# B&R Automation Studio project PLC code - cp (part 14)

#### BRSE_JSON.c
```c
/*! \file BRSE_JSON.c */
/********************************************************************
 * COPYRIGHT -- B&R
 ********************************************************************
 * Library: BRSE_JSON
 * File: BRSE_JSON.c
 * Author: Florian Damerow
 * Created: March 09, 2011
 *******************************************************************/

#include <bur/plctypes.h>
#include "BRSE_JSON.h"
#include <AsBrStr.h>
#include <string.h>
#include "BRSE_JSON_Main.h"
STRING tmpVal[80];

UDINT ValToString(UDINT pv_adresse, UINT pvType){
	switch (pvType) {
		case 1: {
				BOOL *var = (BOOL *)pv_adresse;
				brsitoa((BOOL)*var,(UDINT)&tmpVal);
				break;
				}
		case 2: {
				SINT *var = (SINT *)pv_adresse;
				brsitoa((SINT)*var,(UDINT)&tmpVal);
				break;
				}
		case 3: {
				INT *var = (INT *)pv_adresse;
				brsitoa((INT)*var,(UDINT)&tmpVal);
				break;
				}
		case 4: {
				DINT *var = (DINT *)pv_adresse;
				brsitoa((DINT)*var,(UDINT)&tmpVal);
				break;
				}
		case 5: {
				USINT *var = (USINT *)pv_adresse;
				brsitoa((USINT)*var,(UDINT)&tmpVal);
				break;
				}
		case 6: {
				UINT *var = (UINT *)pv_adresse;
				brsitoa((UINT)*var,(UDINT)&tmpVal);
				break;
				}
		case 7: {
				UDINT *var = (UDINT *)pv_adresse;
				brsitoa((UDINT)*var,(UDINT)&tmpVal);
				break;
				}
		case 8: {
				REAL *var = (REAL *)pv_adresse;
				brsftoa((REAL)*var,(UDINT)&tmpVal);
				break;
				}
		case 9: {
				STRING *var = (STRING *)pv_adresse;
				STRING *tmpBuffer = (STRING *)&tmpVal;
				strcpy(tmpVal,"\"");
				tmpBuffer++;
				strncpy(tmpBuffer,var,(sizeof(tmpVal)-3));
				strcat(tmpVal,"\"");
				break;
				}
		case 11:{
				DINT *var = (DINT *)pv_adresse;
				STRING *tmpBuffer = (STRING *)&tmpVal;
				strcpy(tmpVal,"\"");
				tmpBuffer++;
				brsitoa((DINT)*var,(UDINT)tmpBuffer);
				strcat(tmpVal,"\"");
				break;
				}
		case 12:{
				DINT *var = (DINT *)pv_adresse;
				STRING *tmpBuffer = (STRING *)&tmpVal;
				strcpy(tmpVal,"\"");
				tmpBuffer++;
				brsitoa((DINT)*var,(UDINT)tmpBuffer);
				strcat(tmpVal,"\"");
				break;
				}
		/*case 11:{
				TIME *var = pv_adresse;
				STRING *ptmpValue = &tmpValue;
				strcpy(ptmpValue,"\\/Date(");
				ptmpValue = ptmpValue + 7;
				itoa((DINT)*var,ptmpValue);
				strcat(ptmpValue,")\\/");
				break;
				}
		case 11:{
				DATE_AND_TIME *var = pv_adresse;
				BRSE_DTF_DateTimeFormat_typ format;
				UDINT error;
				error = BRSE_DTF_CreateFormat("YYYY-MM-DD-hh:mm:ss", &format);
				if(error == 0){
					BRSE_DTF_DTToString((DATE_AND_TIME)*var, &format, tmpValue);
				}
				break;
				}
		case 12:{
				TIME *var = pv_adresse;
				STRING *ptmpValue = &tmpValue;
				strcpy(ptmpValue,"\\/Time(");
				ptmpValue = ptmpValue + 7;
				itoa((DINT)*var,ptmpValue);
				strcat(ptmpValue,")\\/");
				break;
				}*/
		default: strcpy(tmpVal,"null");
				 break;
	}
	return (UDINT)tmpVal;
}

/*! \interface JSON_Parse
	\brief parses a JSON message and writes the content to the structure on the PLC

	This function block parses the JSON message and writes the content to the structure on the PLC using PV_xgetadr.\n
	The structure must exist.\n
	\n
	It is possible to parse a long JSON message in several pieces. The message can be split at every point.\n
	It is only possible to parse JSON Objects '{name:content}' \n
	arrays or non objects are NOT supported e.g. '[name:content, name2:content2]' or 'name:content' \n
	\n
	The maximal possible struture name is defined in MAX_STRUCT_NAME_LENGTH_Parse. \n
	That means the whole name e.g. 'Structure.Outer[1].Inner.Test' is limited. \n
	\n
	Entering an object will result in going up with the level by 1 \n
	Entering an array will result in going up with the level by 1 \n
	Entering an struct array will result in going up with the level by 2 \n
	\n
	If pDebug != 0 the whole message will be written there. This will be done with the state for every character.\n
	If pDebug = 0 no Debugging will be performed by the system.\n

	If pVariablesNotFound != 0 all Variables found in the Message, but could not be written on the system are listed here.
	They are represented in a JSON array e.g. '["var1","var2"]'.\n
	If pVariablesNotFound = 0 no output will performed wen variables could not be written.\n
	\n
	The funktion block will be stopped when an error accured.\n
	The function block will not be stopped when a warning accures.\n
	\par Errors:\n
	\arg 1001	invalid JSON in parsestate 0
	\arg 1002	invalid JSON in parsestate 1
	\arg 1003	invalid JSON in parsestate 3
	\arg 1004	invalid JSON in parsestate 4
	\arg 1005	invalid JSON in parsestate 6
	\arg 1006	invalid JSON in parsestate 7
	\arg 1007	Structure depth is deeper than MAX_STRUCT_DEPTH_Parse

	\par Warnings:\n
	\arg 3001	data type not supported
	\arg 3002	variable not found

	\par General: \n
	\arg 2001	parsing so far successful, but end of JSON message net reached yet
	\arg 0		successfuly finished parsing

	\param[in] pMessage Pointer to the JSON Message (String)
	\param[in] pDebug Pointer Debug Buffer (String)
	\param[in] SizeDebug size of the Debug Buffer
	\param[in] pVariablesNotFound Pointer Buffer of VariablesNotFound (String)
	\param[in] SizeVariablesNotFound size of the VariablesNotFound Buffer
	\param[in] MaxLoopIdx used to control cpu load. Allows multiple entries to be parsed each scan.

	\param[out] ErrorInfo contains the Error/Warning/General Codes.
	\param[out] Status signals when block is done=1 or error=2.

*/

void JSON_Parse(struct JSON_Parse* inst)
{
	STRING *pBuff = (STRING *)inst->pMessage;

	UDINT pBuffOld = 0;
	inst->ErrorInfo = 0;

	/* gets the length of the message, only 1 time */
	if(inst->messageLength == 0) {
		inst->messageLength = brsstrlen((UDINT)inst->pMessage);
	}

	if(inst->MaxLoopIdx == 0) {
		inst->MaxLoopIdx = 1000;					// try to set a default value
	}

	/* 	loop index makes it possible to process larger strings, since we don't have to process the whole string in 1 cycle.
			We try to process mutiple variables in 1 cycle.
			If max. loop index is too high we get a cycle time violation.
	*/
	while(inst->buffIdx < inst->messageLength && inst->loopIdx < inst->MaxLoopIdx){			/* while buffer indeex is smaller than length and loop index smaller then max loop index */
		switch(inst->parsestate){
			case 0:
				if(pBuff[inst->buffIdx] == '{'){
					inst->parsestate = 1;
					inst->parselevel++;
					inst->buffIdx++;
					if(inst->pVariablesNotFound != 0 && inst->SizeVariablesNotFound > 2){
						strcpy((STRING *)inst->pVariablesNotFound,"[");
					}
				}
				else if(pBuff[inst->buffIdx] == ' '){
					inst->buffIdx++;
				}
				else{
					inst->ErrorInfo = 1001; /*invalid JSON*/
					inst->Status 	= 2;
					return;
				}
				break;

			case 1:
				if(pBuff[inst->buffIdx] == '"'){
					inst->parsestate = 2;
					inst->buffIdx++;
				}
				else if(pBuff[inst->buffIdx] == ' ' || pBuff[inst->buffIdx] == 9 || pBuff[inst->buffIdx] == 10 || pBuff[inst->buffIdx] == 11 || pBuff[inst->buffIdx] == 12){
					inst->buffIdx++;
				}
				else{
					inst->ErrorInfo = 1002; /*invalid JSON*/
					inst->Status 	= 2;
					return;
				}
				break;

			case 2:
				if(pBuff[inst->buffIdx] != '"'){
					inst->pvName[inst->parselevel][inst->j] = pBuff[inst->buffIdx];
					inst->j++;
					inst->buffIdx++;
				}
				else {
					inst->pvName[inst->parselevel][inst->j] = '\0';
					inst->j = 0;
					inst->parsestate = 3;
					inst->buffIdx++;
				}
				break;

			case 3:
				if(pBuff[inst->buffIdx] == ':'){
					inst->parsestate = 4;
					inst->buffIdx++;
				}
				else if(pBuff[inst->buffIdx] == ' ' || pBuff[inst->buffIdx] == 9 || pBuff[inst->buffIdx] == 10 || pBuff[inst->buffIdx] == 11 || pBuff[inst->buffIdx] == 12){
					inst->buffIdx++;
				}
				else{
					inst->ErrorInfo = 1003; /*invalid JSON*/
					inst->Status 	= 2;
					return;
				}
				break;

			case 4:
				if(pBuff[inst->buffIdx] == '{'){
					inst->parsestate = 1;
					inst->parselevel++;
					inst->buffIdx++;
				}
				else if(pBuff[inst->buffIdx] == '['){
					/*strcat(inst->pvName[inst->parselevel],"[");
					strcat(inst->pvName[inst->parselevel],"0");
					strcat(inst->pvName[inst->parselevel],"]");*/
					inst->isArray[inst->parselevel] = 1;
					inst->parselevel++;
					inst->buffIdx++;
				}
				else if(pBuff[inst->buffIdx] == '\"'){
					inst->Buffer[inst->j] = pBuff[inst->buffIdx];
					inst->buffIdx++;
					inst->j++;
					inst->parsestate = 41;
				}
				else if(pBuff[inst->buffIdx] != '{' && pBuff[inst->buffIdx] != ' ' && pBuff[inst->buffIdx] != '['){ /*maybe better to check for " or - or number*/
					inst->parsestate = 5;
				}
				else if(pBuff[inst->buffIdx] == ' ' || pBuff[inst->buffIdx] == 9 || pBuff[inst->buffIdx] == 10 || pBuff[inst->buffIdx] == 11 || pBuff[inst->buffIdx] == 12){
					inst->buffIdx++;
				}
				else{
					inst->ErrorInfo = 1004; /*invalid JSON*/
					inst->Status 	= 2;
					return;
				}
				break;

			case 41: /* is in String */
				if(pBuff[inst->buffIdx] == '\"'){
					inst->Buffer[inst->j] = pBuff[inst->buffIdx];
					inst->j++;
					inst->Buffer[inst->j] = '\0';
					inst->j=0;
					inst->buffIdx++;
					inst->parsestate = 51;
				}
				else if(pBuff[inst->buffIdx] == '\\'){
					inst->Buffer[inst->j] = pBuff[inst->buffIdx];
					inst->j++;
					inst->buffIdx++;
					inst->Buffer[inst->j] = pBuff[inst->buffIdx];
					inst->j++;
					inst->buffIdx++;
				}
				else{
					inst->Buffer[inst->j] = pBuff[inst->buffIdx];
					inst->j++;
					inst->buffIdx++;
				}
				break;

			case 5:
				if(pBuff[inst->buffIdx] != '}' && pBuff[inst->buffIdx] != ' ' && pBuff[inst->buffIdx] != ',' && pBuff[inst->buffIdx] != ']'){
					inst->Buffer[inst->j] = pBuff[inst->buffIdx];
					inst->j++;
					inst->buffIdx++;
				}
				else{
					STRING mystring[5] = "256";

					UINT myint = strcmp(mystring, inst->Buffer);
					if(myint == 0)
					{
						inst->j = inst->j;
					}
					inst->Buffer[inst->j] = '\0';
					inst->j=0;
					inst->parsestate = 51;
				}
				break;

			case 51: /*write variable*/
				memset((UDINT *)(inst->fullName),0,sizeof(inst->fullName));
				{
					UINT i = 1;
					UDINT adresse;
					UDINT datalen;
					UDINT pvType;
					UDINT pvLength;
					UINT pvStructMembers;
					STRING tmpStr[5];
					while(i <= inst->parselevel && (sizeof(inst->fullName)-strlen(inst->fullName)-7) > strlen(inst->pvName[i])){
						strcat(inst->fullName,inst->pvName[i]);
						if(inst->isArray[i] == 1){
							strcat(inst->fullName,"[");
							brsitoa(inst->pvIndex[i],(UDINT)&tmpStr);
							strcat(inst->fullName,tmpStr);
							strcat(inst->fullName,"]");
						}
						if(i < inst->parselevel && inst->isArray[i] == 0){
							strcat(inst->fullName,".");
						}
						i++;
					}
					inst->ErrorInfo = PV_ninfo((STRING *)&inst->fullName, &pvType, &pvLength, &pvStructMembers);
					if(inst->ErrorInfo == 0){
						inst->ErrorInfo = PV_xgetadr((STRING *)&inst->fullName, &adresse, &datalen);
					}
					else{
						inst->ErrorInfo = 3002; /* variable not found */
					}
					if(inst->ErrorInfo == 0){
						STRING *Buffer = (STRING *)&inst->Buffer;
						if(*Buffer == '\"'){
							Buffer++;
							if(inst->Buffer[strlen(Buffer)] == '\"'){
								inst->Buffer[strlen(Buffer)] = '\0';
							}
						}
						if(strstr(inst->Buffer,"null") == 0){
							switch(pvType){
								case 0:{
									DINT *adr = (DINT *)adresse;
									*adr = (DINT)brsatoi((UDINT)Buffer);
									break;
									}
								case 1:{
										BOOL *adr = (BOOL *)adresse;

										if(strstr(Buffer, "true")){
											*adr = 1;
										}
										else if(strstr(Buffer, "false")){
											*adr = 0;
										}
										else if(brsatoi((UDINT)Buffer) != 0){
											*adr = 1;
										}
										else{
											*adr = 0;
										}
										break;
									}
								case 2:{
									SINT *adr = (SINT *)adresse;
									*adr = (SINT)brsatoi((UDINT)Buffer);
									break;
									}
								case 3:{
									INT *adr = (INT *)adresse;
									*adr = (INT)brsatoi((UDINT)Buffer);
									break;
									}
								case 4:{
									DINT *adr = (DINT *)adresse;
									*adr = (DINT)brsatoi((UDINT)Buffer);
									break;
									}
								case 5:{
									USINT *adr = (USINT *)adresse;
									*adr = (USINT)brsatoi((UDINT)Buffer);
									break;
									}
								case 6:{
									UINT *adr = (UINT *)adresse;
									*adr = (UINT)brsatoi((UDINT)Buffer);
									break;
									}
								case 7:{
									UDINT *adr = (UDINT *)adresse;
									*adr = (UDINT)brsatoi((UDINT)Buffer);
									break;
									}
								case 8:{
									REAL *adr = (REAL *)adresse;
									*adr = (REAL)brsatof((UDINT)Buffer);
									break;
									}
								case 9:{
									STRING *adr = (STRING *)adresse;
									strncpy(adr, Buffer, pvLength-1);
									break;
									}
								case 11:{
									DINT *adr = (DINT *)adresse;
									*adr = (DINT)brsatoi((UDINT)Buffer);
									break;
									}
								case 12:{
									DINT *adr = (DINT *)adresse;
									*adr = (DINT)brsatoi((UDINT)Buffer);
									break;
									}
								case 14:{
										LREAL *adr = (LREAL *)adresse;
										*adr = (LREAL)brsatof((UDINT)Buffer);
										break;
									}
								/*case 11:{
									DINT *adr = adresse;
									STRING *Buffer = &inst->Buffer;
									Buffer = strstr(inst->Buffer,")\\/");
									if(Buffer != 0){
										*Buffer = '\0';
										Buffer = strstr(inst->Buffer,"\\/Date(");
										if(Buffer != 0){
											Buffer = Buffer + 7;
										}
									}
									*adr = (DINT)atoi(Buffer);
									break;
									}
								case 12:{
									DINT *adr = adresse;
									STRING *Buffer = &inst->Buffer;
									Buffer = strstr(inst->Buffer,")\\/");
									if(Buffer != 0){
										*Buffer = '\0';
										Buffer = strstr(inst->Buffer,"\\/Time(");
										if(Buffer != 0){
											Buffer = Buffer + 7;
										}
									}
									*adr = (DINT)atoi(Buffer);
									break;
									}*/

								default:{
									inst->ErrorInfo = 3001;
									break;
									}
							}
						}
					}
					else{
						inst->ErrorInfo = 3002; /* variable not found */
						if(inst->pVariablesNotFound != 0 && inst->SizeVariablesNotFound != 0){
							if((inst->SizeVariablesNotFound - strlen((STRING *)inst->pVariablesNotFound)-2) > strlen(inst->fullName)+3){
								if(strlen((STRING *)inst->pVariablesNotFound) > 2){
									strcat((STRING *)inst->pVariablesNotFound,",");
								}
								strcat((STRING *)inst->pVariablesNotFound,"\"");
								strcat((STRING *)inst->pVariablesNotFound,inst->fullName);
								strcat((STRING *)inst->pVariablesNotFound,"\"");
							}
						}
					}
					if(pBuff[inst->buffIdx] == ',' && inst->isArray[inst->parselevel-1] == 1){
						inst->buffIdx++;
						inst->pvIndex[inst->parselevel-1]++;
						inst->parsestate = 4;
					}
					else{
						inst->parsestate = 6;
					}
				}
				break;

			case 6:
				if(pBuff[inst->buffIdx] == '}'){
					inst->parsestate = 6;
					inst->pvIndex[inst->parselevel-1] = 0;
					strcpy(inst->pvName[inst->parselevel],"");	// if the string is not cleared, the parseing is not working right - olsenm
					inst->parselevel--;
					inst->buffIdx++;
				}
				else if(pBuff[inst->buffIdx] == ']'){
					inst->parsestate = 6;
					inst->pvIndex[inst->parselevel-1] = 0;
					strcpy(inst->pvName[inst->parselevel],"");	// if the string is not cleared, the parseing is not working right - olsenm
					inst->parselevel--;
					inst->isArray[inst->parselevel] = 0;
					inst->buffIdx++;
				}
				else if(pBuff[inst->buffIdx] == ','){
					inst->parsestate = 7;
					inst->pvIndex[inst->parselevel-1]++;
					inst->buffIdx++;
				}
				else if(pBuff[inst->buffIdx] == ' ' || pBuff[inst->buffIdx] == 9 || pBuff[inst->buffIdx] == 10 || pBuff[inst->buffIdx] == 11 || pBuff[inst->buffIdx] == 12){
					inst->buffIdx++;
				}
				else{
					inst->ErrorInfo = 1005; /*invalid JSON*/
					inst->Status 	= 2;
					return;
				}
				break;

			case 7:
				if(pBuff[inst->buffIdx] == '{'){
					inst->parselevel++;
					inst->parsestate = 1;
					inst->buffIdx++;
				}
				else if(pBuff[inst->buffIdx] == '\"'){
					inst->parsestate = 1;
				}
				else if(pBuff[inst->buffIdx] == ' ' || pBuff[inst->buffIdx] == 9 || pBuff[inst->buffIdx] == 10 || pBuff[inst->buffIdx] == 11 || pBuff[inst->buffIdx] == 12){
					inst->buffIdx++;
				}
				else{
					inst->ErrorInfo = 1006; /*invalid JSON*/
					inst->Status 	= 2;
					return;
				}
		}

		/* DEBUGGING */
		if(inst->pDebug != 0){
			if(pBuffOld != pBuff[inst->buffIdx]){
				STRING BUFFER2[4];
				STRING BUFFER3[2];
				if((inst->SizeDebug - strlen((STRING *)inst->pDebug) - 1) > 7){
					if(inst->parsestateold != inst->parsestate){
						inst->parsestateold = inst->parsestate;
						brsitoa((DINT)inst->parsestate,(UDINT)&BUFFER2);
						strcat((STRING *)inst->pDebug,"(");
						strcat((STRING *)inst->pDebug,BUFFER2);
						strcat((STRING *)inst->pDebug,")");
					}
					BUFFER3[0] = pBuff[inst->buffIdx];
					BUFFER3[1] = 0;
					strcat((STRING *)inst->pDebug,BUFFER3);
				}
			}
			pBuffOld = pBuff[inst->buffIdx];
		}
		inst->loopIdx++;			// loop index counter
	}
	inst->loopIdx = 0;		// reset loop index

	/* Error Handling */
	if(inst->parselevel > MAX_STRUCT_DEPTH_Parse){
		inst->ErrorInfo = 1007;
	}
	if(inst->ErrorInfo >= 1000 && inst->ErrorInfo  < 2000){
		inst->parselevel = 0;
		inst->parsestate = 0;
		memset(inst->pvIndex,0,sizeof(inst->pvIndex));
		memset(inst->pvName,0,sizeof(inst->pvName));
	}
	else if(inst->parselevel != 0){
		inst->ErrorInfo = 2001; /*not done*/
	}
	else{
		if(inst->pVariablesNotFound != 0){
			strcat((STRING *)inst->pVariablesNotFound,"]");
		}
		inst->parsestate = 0;
	}

	/*Status output*/
	if(inst->buffIdx >= inst->messageLength)
	{
		if(inst->ErrorInfo > 0)
		{
			//Done, Error present.
			inst->Status = 2;
		}
		else
		{
			//Done, no errors present.
			inst->Status = 1;
		}

	}
}

/*! \interface JSON_Stringify
	\brief converts a PV variable and the whole structure into a JSON Object using PV_ninfo.

	This function block converts the whole structure of a PV variable into a JSON Object using PV_ninfo. \n
	The variable name should be the same as using the PV_ninfo function. By that it is possible to access any kind of PV variables.\n
	The output is always a JSON object. e.g. '{"varname": ... }' \n
	\n
	The function block has to be run several times until the Status = 1. \n
	Every time the function block is called it creates the JSON output for one new variable inside the Structure. \n
	If the variable in the structure is an array of a non object type the whole array will be created in Output.\n
	\n
	The maximum Output length is defined by MAX_OUTPUT_LENGTH_Stringify.\n
	The maximum Value of a nun array, non structure variable is 80. So Strings are only supported up the 80 characters.\n
	\n
	By using pMessage and MaxLoopIndex multiple entries can be stringified in one scan.\n
	The complete json string is written directly to the buffer pMessage is pointing to.\n

	\par Status Codes:\n
	\arg 1001 Variable not found
	\arg 1002 Variable value too long
	\arg 1003 pStName = 0, zero pointer
	\arg 1 stringify process completed
	\arg 0 stringify process not completet yet - run again

	\param[in] pStName Pointer to the requested variable name
	\param[in] pMessage pointer to output buffer where the entire JSON_String is written.
	\param[in] MaxLoopIndex used to control cpu load. Allows multiple entries to be stringified each scan.

	\param[out] Status returns the Status codes
	\param[out] Output contains the content of one step

*/
void JSON_Stringify(struct JSON_Stringify* inst)
{
	/*
			the loop index makes it possible to process mutiple variables in one cycle
			if the maxloopisx is too high we get a cycle time violation
	*/

	if(inst->MaxLoopIdx == 0) {
		inst->MaxLoopIdx = 100;			// default value
	}

	memset(inst->Output,0,sizeof(inst->Output));

	for(inst->loopIdx = 0; inst->loopIdx < inst->MaxLoopIdx; inst->loopIdx++) {
		STRING *pBuff = 0;
		STRING strBuff[20];
		inst->TaskDoc.Input.StructDepth = MAX_STRUCT_DEPTH_Stringify;

		/*gather information of the structure item*/
		memset(inst->tmpStruct,0,sizeof(inst->tmpStruct));

		if(inst->pStName != 0 )
		{
			strcpy(inst->tmpStruct,(STRING *)inst->pStName);
		}
		else
		{
			inst->Status = 1003;
			return;
		}

		strcat(inst->tmpStruct, inst->pvName[0]);
		for( inst->i = 1; inst->i <= inst->pvLevel; inst->i++ ){
			if(inst->isArray[inst->i-1] == 0){
				strcat(inst->tmpStruct, ".");
				strcat(inst->tmpStruct, inst->pvName[inst->i]);
			}
			else{
				inst->isArray[inst->pvLevel] = 1;
				strcat(inst->tmpStruct,"[");
				brsitoa(inst->pvIndex[inst->i-1],(UDINT)&strBuff);
				strcat(inst->tmpStruct,strBuff);
				strcat(inst->tmpStruct,"]");
			}
		}
		/*Search in PV-list*/
		inst->TaskDoc.Output.StatusInfo = PV_ninfo((STRING *)&inst->tmpStruct, &inst->pvType, &inst->pvLength, &inst->pvStructMembers[inst->pvLevel]);
		if(inst->pvType == 0){
			STRING name[80];
			inst->TaskDoc.Output.StatusSearch = PV_item((STRING *)&inst->tmpStruct, 0, (STRING *)&name);
			if(inst->TaskDoc.Output.StatusSearch != 0){
				inst->pvType = 4;
				inst->pvStructMembers[inst->pvLevel] = 1;
				inst->TaskDoc.Output.StatusSearch = 0;
			}
		}
		if(inst->pvType == 15){
			inst->isArray[inst->pvLevel] = 1;
			strcat(inst->tmpStruct,"[");
			brsitoa(inst->pvIndex[inst->pvLevel],(UDINT)&strBuff);
			strcat(inst->tmpStruct,strBuff);
			strcat(inst->tmpStruct,"]");
			inst->pvLevel = inst->pvLevel + 1;
			inst->TaskDoc.Output.StatusInfo = PV_ninfo((STRING *)&inst->tmpStruct, &inst->pvType, &inst->pvLength, &inst->pvStructMembers[inst->pvLevel]);
		}
		else{
			inst->isArray[inst->pvLevel] = 0;
		}
		if( inst->TaskDoc.Output.StatusInfo == 0 ){
			inst->TaskDoc.Output.StatusInfo = PV_xgetadr((STRING *)&inst->tmpStruct,&inst->pv_adresse,&inst->data_len);
		}
		if( inst->TaskDoc.Output.StatusInfo == 0 ){
		/*variable was found*/
			STRING *ValToStr;
			UDINT Size=0;
			memset(inst->tmpValue,0,sizeof(inst->tmpValue));
			if(inst->pvStructMembers[inst->pvLevel]>1){
				strcat(inst->tmpValue,"[");
			}
			ValToStr = (STRING *)ValToString(inst->pv_adresse, inst->pvType);
			if((sizeof(inst->tmpValue)-strlen(inst->tmpValue)-2) > strlen(ValToStr)){
				strcat(inst->tmpValue, ValToStr);
			}
			inst->arrIndex = 1;
			Size = (UDINT)(inst->data_len/inst->pvStructMembers[inst->pvLevel]);
			pBuff = (STRING *)((UDINT)inst->pv_adresse+Size);
			/*build array output */
			while(inst->arrIndex < inst->pvStructMembers[inst->pvLevel]){
				ValToStr = (STRING *)ValToString((UDINT)pBuff, inst->pvType);
				if((sizeof(inst->tmpValue)-strlen(inst->tmpValue)-2) <= strlen(ValToStr)){
					inst->Status = 1002; /*Variable Value too long*/
					return;
				}
				strcat(inst->tmpValue, ",");
				strcat(inst->tmpValue, ValToStr);
				pBuff = pBuff+Size;
				inst->arrIndex++;
			}
			if(inst->pvStructMembers[inst->pvLevel]>1){
				strcat(inst->tmpValue,"]");
			}

			/*get inner variable name*/
			pBuff = (inst->tmpStruct)+strlen(inst->tmpStruct);
			while((UDINT)pBuff >= (UDINT)&(inst->tmpStruct) && *pBuff != '.'){
				pBuff--;
			}
			pBuff++;
			/*create JSON output*/
			//memset(inst->Output,0,sizeof(inst->Output)); Memset should be done outside for loop. Or output will just contain the latest iteration output. Valdtp V1.11.0
			if((43+strlen(inst->tmpValue)) > sizeof(inst->Output)){
				inst->Status = 1002; /*Variable Value too long*/
				return;
			}
			if(!(inst->isArray[inst->pvLevel-1] == 1 && inst->pvIndex[inst->pvLevel-1] > 0)){
				if((inst->pvLevel == 0 && inst->pvIndex[0] == 0) || (inst->isArray[inst->pvLevel-1] == 1 && (inst->pvLevel-1) == 0) ){
					strcat(inst->Output, "{");

				}
				strcat(inst->Output, "\"");
				if( inst->pvLevel == 0){
					strcat(inst->Output, (STRING *)inst->pStName);
				}
				else if(inst->isArray[inst->pvLevel-1] == 1){
					if((inst->pvLevel-1) > 0){
						strcat(inst->Output, inst->pvName[inst->pvLevel-1]);
					}
					else{
						strcat(inst->Output, (STRING *)inst->pStName);
					}
				}else{
					strcat(inst->Output, inst->pvName[inst->pvLevel]);
				}
				strcat(inst->Output, "\":");
				if(inst->isArray[inst->pvLevel-1]){
					strcat(inst->Output, "[");
				}
			}
			if( inst->pvType == 0 ){
				strcat(inst->Output, "{");
			}
			if( inst->pvType != 0 && inst->pvType != 15 ){
				strcat(inst->Output, inst->tmpValue);
			}

			inst->pvSearchComplete = 0;

			if( (inst->pvType == 0) && (inst->pvLevel < (inst->TaskDoc.Input.StructDepth-1)) ){
				/*variable is a structure and its ok to go look inside it*/
				/*ok. proceed to next level.*/
				inst->TaskDoc.Output.StatusSearch = PV_item((STRING *)&inst->tmpStruct, inst->pvIndex[inst->pvLevel], (STRING *)&inst->pvName[inst->pvLevel+1]);
				inst->pvLevel = inst->pvLevel + 1;
			}
			else if( (inst->pvLevel > 0) || (inst->pvLevel==0 && inst->pvIndex[inst->pvLevel] < (inst->pvStructMembers[inst->pvLevel]))){ /*..in case its 0 we have a problem*/
			/*variable is a basic datatype*/
				do{
					inst->pvContinue = 0;
					if( inst->isArray[inst->pvLevel-1] == 1){
						if( inst->pvIndex[inst->pvLevel-1] < (inst->pvStructMembers[inst->pvLevel-1]-1)){
							/*ok. take the next item in prior structure*/
							inst->pvIndex[inst->pvLevel-1] = inst->pvIndex[inst->pvLevel-1] + 1;
							strcpy(inst->pvName[inst->pvLevel],"");		// if the string is not cleared, the stringify is not working right - olsenm
							inst->pvLevel = inst->pvLevel - 1;

							strcat(inst->Output, ",");
							break; /*..from loop*/
						}
						else{
							strcat(inst->Output, "]");
							strcpy(inst->pvName[inst->pvLevel],"");		// if the string is not cleared, the stringify is not working right - olsenm
							inst->pvLevel = inst->pvLevel - 1;
							inst->pvIndex[inst->pvLevel] = 0;
							if( inst->pvLevel > 0 ){
								inst->pvContinue = 1;
							}else{
								inst->pvSearchComplete = 1;
								strcat(inst->Output, "}");
								break;
							}
						}
					}
					else{
						if( inst->pvIndex[inst->pvLevel-1] < (inst->pvStructMembers[inst->pvLevel-1]-1)){
							/*ok. take the next item in prior structure*/
							inst->pvIndex[inst->pvLevel-1] = inst->pvIndex[inst->pvLevel-1] + 1;
							strcat(inst->Output, ",");
							break; /*..from loop*/
						}else{
							/*continue looking in the prior structure if the index is smaller members*/
							strcpy(inst->pvName[inst->pvLevel],"");																		// if the string is not cleared, the stringify is not working right - olsenm
							inst->pvLevel = inst->pvLevel - 1;
							if(inst->pvLevel>=0){
								strcat(inst->Output, "}");
							}
							inst->pvIndex[inst->pvLevel] = 0; /*this one is used the nest time a structure is found on this level*/
							if( inst->pvLevel > 0 ){
								inst->pvContinue = 1;
							}else{
								inst->pvSearchComplete = 1;
								strcat(inst->Output, "}");
								break;
							}
						}
					}
				}
				while(inst->pvContinue != 0);

				/*look after following member in prior structure*/
				if( inst->pvLevel > 0 ){
					strcpy(inst->tmpStruct,(STRING *)inst->pStName);

					strcat(inst->tmpStruct, inst->pvName[0]);
					for( inst->i = 1; inst->i <= (inst->pvLevel-1); inst->i++ ){
						if(strlen(inst->pvName[inst->i]) != 0){
							strcat(inst->tmpStruct, ".");
							strcat(inst->tmpStruct, inst->pvName[inst->i]);
						}
					}
					/*ok. get the next variable*/
					inst->TaskDoc.Output.StatusSearch = PV_item((STRING *)&inst->tmpStruct, inst->pvIndex[inst->pvLevel-1], (STRING *)&inst->pvName[inst->pvLevel]);
				}else if((inst->pvLevel==0 && inst->pvIndex[inst->pvLevel] == (inst->pvStructMembers[inst->pvLevel]))){
					/*no more items in top structure*/
					inst->pvSearchComplete = 1;
				}
			}else{
				inst->pvSearchComplete = 1;
			}
			if(inst->pvSearchComplete == 1){
				inst->Status = 1;
			}else{
				inst->Status = 0;
			}
		}else{
			 inst->Status = 1001; /*variable not found*/
		}

		if(inst->Status == 1) {
			break; 									// break out of for loop because the function block is done processing the variables
		}

	}//END FOR

	/*Must always check that pointers are != 0 or it will krasch PLC. Valdtp V1.11.0*/
	if(inst->pMessage != 0)
	{
		/*
			instead of copying the output outside the fb we do in inside, so we can process mutiple variables in 1 cycle  -olsenm
		*/
		UDINT outLen = brsstrlen((UDINT)inst->Output);// length of the generated output string
		UDINT tmpMsgPtr = (UDINT)&((char*)inst->pMessage)[inst->messageIdx];	// pointer to where the output can be copied to
		strcpy((char*)tmpMsgPtr,inst->Output);									// copy the string
		inst->messageIdx += outLen;		// messageidx keeps track of where in the message string we can copy the output string

	}

}
```

#### version_history.c
```c
/*!\file version_history.c */

/*!
	\page History
	\section History

	\par V1.00.0
		\arg First version created

	\par V1.00.1
		\arg Helpfile and example added.

	\par V1.01.0
		\arg Helpfile updated
		\arg First release version.

	\par V1.02.0
		\arg Helpfile updated

	\par V1.10.0
		\arg Library dependency changed from AsString to AsBrStr.
             Add #include <AsBrStr.h>
        \arg Functions atof, ftoa, atoi and itoa are changed to brsatof, brsftoa, brsatoi, and brsitoa
             to avoid name conflict.
        \arg Functions strcat and strcpy can continue to be used from string.h
	\par V1.11.0
		\arg Library updated, changed command structure for functions. Improving usage with large data amounts.
			 Possible to set number of iterations run per scan.
			 Output directly into an output buffer has beeen added making it possible to stringify several entries in one scan.

		\arg Examples replaced and simplified. Package that is imported instead of an entire project.
			 The simplification should make the javascript code and example tasks easier to understand.
			 TestProgram task added.
	\par V1.12.0
		\arg Added support for ASCII charaters 9 -> 12. TAB, New Line, Vertical Tab and New page.
			 Have the same effect has an blank space ' '.
			 This to ease the usage of third party software like Notepad++ for editing of the JSON string.
*/
```

### MTFilter.var
```iecst
(*Error*)
VAR CONSTANT
	mtBCD_ERR_FILTER_TYPE_INVALID : DINT := -1058012158; (*Filter type is invalid.*)
	mtBCD_ERR_FILTER_ORDER_INVALID : DINT := -1058012157; (*Filter order is invalid.*)
	mtBCD_ERR_CUTOFF_FREQ_INVALID : DINT := -1058012156; (*Cutoff frequency of the filter is invalid.*)
	mtBCD_ERR_CENTER_FREQ_INVALID : DINT := -1058012155; (*Center frequency of the filter is invalid.*)
	mtBCD_ERR_FILTER_BANDWIDTH : DINT := -1058012154; (*Bandwidth of the filter is invalid.*)
	mtBCD_ERR_FREQ_NUM_INVALID : DINT := -1058012153; (*Filter frequency of the numerator is invalid.*)
	mtBCD_ERR_DAMPING_NUM_INVALID : DINT := -1058012152; (*Damping of the numerator is invalid.*)
	mtBCD_ERR_FREQ_DEN_INVALID : DINT := -1058012151; (*Filter frequency of the denominator is invalid.*)
	mtBCD_ERR_DAMPING_DEN_INVALID : DINT := -1058012150; (*Damping of the denominator is invalid.*)
	mtBCD_ERR_FILTER_WINDOW_INVALID : DINT := -1058012149; (*Window length of the filter is invalid.*)
	mtBCD_ERR_TRANSFER_FCN_INVALID : DINT := -1058012148; (*Transfer function (Numerator or Denominator) of the FB MTFilterKalman is invalid.*)
	mtBCD_ERR_NOISEREDUCTION_INVALID : DINT := -1058012147; (*The parameter NoiseReduction of the FB MTFilterKalman is invalid.*)
	mtBCD_ERR_DISTURB_MODEL_INVALID : DINT := -1058012146; (*The disturbance model of the FB MTFilterKalman is invalid.*)
END_VAR
(*Warning*)
VAR CONSTANT
	mtBCD_WRN_FILTER_TYPE_INVALID : DINT := -2131753982; (*Filter type is invalid.*)
	mtBCD_WRN_FILTER_ORDER_INVALID : DINT := -2131753981; (*Filter order is invalid.*)
	mtBCD_WRN_CUTOFF_FREQ_INVALID : DINT := -2131753980; (*Cutoff frequency of the filter is invalid.*)
	mtBCD_WRN_CENTER_FREQ_INVALID : DINT := -2131753979; (*Center frequency of the filter is invalid.*)
	mtBCD_WRN_FILTER_BANDWIDTH : DINT := -2131753978; (*Bandwidth of the filter is invalid. *)
	mtBCD_WRN_FREQ_NUM_INVALID : DINT := -2131753977; (*Filter frequency of the numerator is invalid. *)
	mtBCD_WRN_DAMPING_NUM_INVALID : DINT := -2131753976; (*Damping of the numerator is invalid. *)
	mtBCD_WRN_FREQ_DEN_INVALID : DINT := -2131753975; (*Filter frequency of the denominator is invalid. *)
	mtBCD_WRN_DAMPING_DEN_INVALID : DINT := -2131753974; (*Damping of the denominator is invalid. *)
	mtBCD_WRN_FILTER_WINDOW_INVALID : DINT := -2131753973; (*Window length of the filter is invalid. *)
	mtBCD_WRN_TRANSFER_FCN_INVALID : DINT := -2131753972; (*Transfer function (Numerator or Denominator) of the FB MTFilterKalman is invalid.*)
	mtBCD_WRN_NOISEREDUCTION_INVALID : DINT := -2131753971; (*The parameter NoiseReduction of the FB MTFilterKalman is invalid.*)
	mtBCD_WRN_DISTURB_MODEL_INVALID : DINT := -2131753970; (*The disturbance model of the FB MTFilterKalman is invalid.*)
END_VAR
```

### Program Logical/LineCtrl/LineCtrl (IEC)

#### Configuration.st
```iecst
ACTION Configuration:

	// Update ancillaries status used
	xPrimerStopped := PrimerStopped(ADR(Primer));

	//Line's ancillaries assignation//
	//Feeder
	//Parameters
	Feeder.Parameters.xSimulationMode 				:= gMachine.Pt.ConfigNameID = GC_CONFIG_SIMTEST_ID;
	Feeder.Parameters.xLineInAuto 					:= gMachine.St.Mode.xAuto;
	Feeder.Parameters.Media 						:= gMachine.parSw.Media;
	Feeder.Parameters.rBeltSpeedSetPoint 			:= MAX(1, Belt.parameters.rSetPointSpeed);
	Feeder.Parameters.iCentralOffset 				:= Feeder.ParSw.iCentralOffset;
	Feeder.Parameters.iCounterSetPointL1 			:= UDINT_TO_INT(gMachine.parSw.iNumCopies AND 16#FFFF);
	Feeder.Parameters.iCounterSetPointL2 			:= UDINT_TO_INT(SHR((gMachine.parSw.iNumCopies AND 16#F0000),16));
	IF NOT gMachine.parSw.Dtp.xDoubleLine THEN
		Feeder.Parameters.iLineConfig:= 0;
	ELSE
		Feeder.Parameters.iLineConfig:= 2;
	END_IF
	Feeder.Parameters.LineState						:= gLine.Status;
	Feeder.Parameters.LineStatusSummary				:= gLine.StatusSummary;

	//Commands
	Feeder.Commands.xResetAlarms := gMachine.AutoCmd.xReset OR gLine.Commands.Print;
	Feeder.Commands.xNewOrder := EDGEPOS(gMachine.St.xRobotReadyToPrint);

	//Primer
	//Parameters
	Primer.Parameters.xSimulationMode 				:= gMachine.Pt.ConfigNameID = GC_CONFIG_SIMTEST_ID;
	Primer.Parameters.xLineInAuto 					:= gMachine.St.Mode.xAuto;
	Primer.Parameters.Media 						:= gMachine.parSw.Media;
	Primer.Parameters.rBeltSpeedSetPoint 			:= MAX(1, Belt.parameters.rSetPointSpeed);
	Primer.Parameters.xDoubleLine 					:= gMachine.parSw.Dtp.xDoubleLine;
	Primer.Parameters.LineState						:= gLine.Status;
	Primer.Parameters.LineStatusSummary				:= gLine.StatusSummary;
	Primer.Parameters.rMediaLength 					:= gMachine.parSw.Media.rLength;
	Primer.Parameters.rSpeedSetPoint 				:= Belt.parameters.rSetPointSpeed;
	Primer.Parameters.xPreviousDeviceStopped 		:= NOT Feeder.Status.Device.xFeeding;

	//Commands
	Primer.Commands.xResetAlarms 					:= gMachine.AutoCmd.xReset;
	Primer.Commands.xEnteringMedia 					:= gFeeder.Status.Device.xFeeding;

	//SARM
	//Parameters
	Sarm.Parameters.xSimulationMode 				:= gMachine.Pt.ConfigNameID = GC_CONFIG_SIMTEST_ID;
	Sarm.Parameters.xLineInAuto 					:= gMachine.St.Mode.xAuto;
	Sarm.Parameters.Media 							:= gMachine.parSw.Media;
	Sarm.Parameters.xDoubleLine 					:= gMachine.parSw.Dtp.xDoubleLine;
	Sarm.Parameters.LineState						:= gLine.Status;
	Sarm.Parameters.rMediaLength 					:= gMachine.parSw.Media.rLength;
	Sarm.Parameters.rSpeedSetPoint 					:= Belt.parameters.rSetPointSpeed;

	Sarm.Parameters.xPreviousDeviceEmpty 			:= (xPrimerEmptied OR xPrimerStopped OR (NOT Feeder.Status.Device.xFeeding AND Feeder.Parameters.xInstalled AND NOT Primer.Parameters.xInstalled)) ;
	IF NOT gMachine.parSw.Dtp.xDoubleLine THEN
		Sarm.Parameters.iLineConfig:= 0;
	ELSE
		Sarm.Parameters.iLineConfig:= 2;
	END_IF
	//Commands
	Sarm.Commands.xResetAlarms 						:= gMachine.AutoCmd.xReset;

	//Dryer
	//Parameters
	Dryer.Parameters.xLineInAuto 					:= gMachine.St.Mode.xAuto;
	Dryer.Parameters.Hw.rDryerLength 				:= 5000.0;
	Dryer.Parameters.rSpeedSetPoint 				:= Belt.parameters.rSetPointSpeed;
	Dryer.Parameters.rMediaLength 					:= gMachine.parSw.Media.rLength;
	Dryer.Parameters.rMediaWidth 					:= gMachine.parSw.Media.rWidth;
	Dryer.Parameters.rMediaThickness 				:= gMachine.parSw.Media.rThickness;
	Dryer.Parameters.rMediaGap 						:= gMachine.parSw.Media.rGap;
	Dryer.Parameters.LineState 						:= Line.Status;
	Dryer.Parameters.rDocumentWidth 				:= gMachine.parSw.Document.rWidth;
	Dryer.Parameters.rDocumentLength 				:= gMachine.parSw.Document.rLength;
	Dryer.Parameters.rDocumentOffsetL1				:= gMachine.parSw.Document.rOffsetL1; //NOZDRYER-467
	Dryer.Parameters.rDocumentOffsetL2				:= gMachine.parSw.Document.rOffsetL2; //NOZDRYER-467
	Dryer.Parameters.xDoubleLine 					:= gMachine.parSw.Dtp.xDoubleLine;
	//Commands
	Dryer.Commands.xResetAlarms 					:= gMachine.AutoCmd.xReset;

	//OverPrimer
	//Parameters
	OverVarnish.Parameters.xSimulationMode 		:= gMachine.Pt.ConfigNameID = GC_CONFIG_SIMTEST_ID;
	OverVarnish.Parameters.xLineInAuto 			:= gMachine.St.Mode.xAuto;
	OverVarnish.Parameters.Media 				:= gMachine.parSw.Media;
	OverVarnish.Parameters.xDoubleLine 			:= gMachine.parSw.Dtp.xDoubleLine;
	OverVarnish.Parameters.LineState			:= gLine.Status;
	OverVarnish.Parameters.LineStatusSummary	:= gLine.StatusSummary;
	OverVarnish.Parameters.rMediaLength 		:= gMachine.parSw.Media.rLength;
	OverVarnish.Parameters.rSpeedSetPoint	:= MAX(1, Belt.parameters.rSetPointSpeed);
	OverVarnish.Parameters.xPreviousDeviceStopped := ThickCtrl.status.Belt.xBeltEmpty AND (Dryer.Status.xBeltEmpty OR NOT Dryer.ParSw.xEnabled);

	//Commands
	OverVarnish.Commands.xResetAlarms 				:= gMachine.AutoCmd.xReset;
	OverVarnish.Commands.xEnteringMedia 			:= 	gFeeder.Status.Device.xFeeding OR
														NOT xPrimerEmptied OR
														NOT xSarmEmptied OR
														NOT ThickCtrl.status.Belt.xBeltEmpty OR
														NOT xDryerEmptied;

	//Stacker
	//Parameters
	Stacker.Parameters.xSimulationMode 				:= gMachine.Pt.ConfigNameID = GC_CONFIG_SIMTEST_ID;
	Stacker.Parameters.xLineInAuto 					:= gMachine.St.Mode.xAuto;
	Stacker.Parameters.Media 						:= gMachine.parSw.Media;
	Stacker.Parameters.rSpeedSetPoint	 			:= MAX(1, Belt.parameters.rSetPointSpeed);
	Stacker.Parameters.xDoubleLine 					:= gMachine.parSw.Dtp.xDoubleLine;
	Stacker.Parameters.LineState					:= gLine.Status;
	Stacker.Parameters.LineStatusSummary			:= gLine.StatusSummary;
	Stacker.Parameters.xPreviousDeviceStopped		:= 	ThickCtrl.status.Belt.xBeltEmpty AND
														(Dryer.Status.xBeltEmpty OR NOT Dryer.ParSw.xEnabled) AND
														(OverVarnish.Status.xBeltEmpty OR NOT OverVarnish.ParSw.xEnabled);

	IF Machine.St.HwData.xIsWater THEN
		Stacker.Orders.xHoldReject := gThicknessCtrl.Outputs.xHoldReject OR Line.StatusSummary.xEmptyingBelts;
	ELSE
		Stacker.Orders.xHoldReject := gThicknessCtrl.Outputs.xHoldReject;
	END_IF

	//Commands
	Stacker.Commands.xResetAlarms := gMachine.AutoCmd.xReset;

	//Line media limits
	DefineMediaLimits;

	//Line speed limits
	DefineSpeedLimits;

	//Line features allowed
	DefineLineFeaturesAllowed;

END_ACTION

ACTION DefineMediaLimits:

	iFeederMediaWidth := FeederMaxMediaWidth(ADR(Feeder), ADR(gMachine));
	iFeederMediaLength := FeederMaxMediaLength(ADR(Feeder), ADR(gMachine));
	iFeederMinMediaThickness := FeederMinMediaThickness(ADR(Feeder), ADR(gMachine));
	iFeederMaxMediaThickness := FeederMaxMediaThickness(ADR(Feeder), ADR(gMachine));

	iPrimerMediaWidth := PrimerMaxMediaWidth(ADR(Primer), ADR(gMachine));
	iPrimerMediaLength := PrimerMaxMediaLength(ADR(Primer), ADR(gMachine));
	iPrimerMinMediaThickness := PrimerMinMediaThickness(ADR(Primer), ADR(gMachine));
	iPrimerMaxMediaThickness := PrimerMaxMediaThickness(ADR(Primer), ADR(gMachine));

	iSarmMediaWidth := SarmMaxMediaWidth(ADR(Sarm), ADR(gMachine));
	iSarmMediaLength := SarmMaxMediaLength(ADR(Sarm), ADR(gMachine));
	iSarmMinMediaThickness := SarmMinMediaThickness(ADR(Sarm), ADR(gMachine));
	iSarmMaxMediaThickness := SarmMaxMediaThickness(ADR(Sarm), ADR(gMachine));

	iDryerMediaWidth := DryerMaxMediaWidth(ADR(Dryer), ADR(gMachine));
	iDryerMediaLength := DryerMaxMediaLength(ADR(Dryer), ADR(gMachine));
//	iDryerMinMediaThickness := DryerMinMediaThickness(ADR(Dryer), ADR(gMachine));
//	iDryerMaxMediaThickness := DryerMaxMediaThickness(ADR(Dryer), ADR(gMachine));

	iOvervarnishMediaWidth := OvervarnishMaxMediaWidth(ADR(OverVarnish), ADR(gMachine));
	iOvervarnishMediaLength := OvervarnishMaxMediaLength(ADR(OverVarnish), ADR(gMachine));
	iOverVarnishMinMediaThickness := OverVarnishMinMediaThickness(ADR(OverVarnish), ADR(gMachine));
	iOverVarnishMaxMediaThickness := OverVarnishMaxMediaThickness(ADR(OverVarnish), ADR(gMachine));

	iStackerMediaWidth := StackerMaxMediaWidth(ADR(Stacker), ADR(gMachine));
	iStackerMediaLength := StackerMaxMediaLength(ADR(Stacker), ADR(gMachine));
	iStackerMinMediaThickness := StackerMinMediaThickness(ADR(Stacker), ADR(gMachine));
	iStackerMaxMediaThickness := StackerMaxMediaThickness(ADR(Stacker), ADR(gMachine));

	gMachine.Pt.Media.iMaxMediaWidth := MIN(iFeederMediaWidth, iPrimerMediaWidth, iSarmMediaWidth, gMachine.Pt.Hw.iWidth, iDryerMediaWidth, iOvervarnishMediaWidth, iStackerMediaWidth);
	gMachine.Pt.Media.iMaxMediaLength := MIN(iFeederMediaLength, iPrimerMediaLength, iSarmMediaLength, gMachine.parSw.Hw.iMaxMediaLength, iDryerMediaLength, iOvervarnishMediaLength, iStackerMediaLength);
	gMachine.Pt.Media.rMaxMediaThickness := UINT_TO_REAL((MIN(iFeederMaxMediaThickness, iPrimerMaxMediaThickness, iSarmMaxMediaThickness, REAL_TO_UINT(gMachine.Pt.CT.rMaxTicknessMedia*10), iOverVarnishMaxMediaThickness, iStackerMaxMediaThickness)))/10;
	gMachine.Pt.Media.rMinMediaThickness := UINT_TO_REAL((MAX(iFeederMinMediaThickness, iPrimerMinMediaThickness, iSarmMinMediaThickness, REAL_TO_UINT(gMachine.Pt.CT.rMinTicknessMedia*10), iOverVarnishMinMediaThickness, iStackerMinMediaThickness)))/10;
END_ACTION

ACTION DefineSpeedLimits:

	rFeederMaxSpeed := FeederMaxSpeed(ADR(Feeder), ADR(gBelt));
	rPrimerMaxSpeed := PrimerMaxSpeed(ADR(Primer), ADR(gBelt));
	rSarmMaxSpeed := SarmMaxSpeed(ADR(Sarm), ADR(gBelt));
	rDryerMaxSpeed := DryerMaxSpeed(ADR(Dryer), ADR(gBelt));
	rOvervarnishMaxSpeed := OvervarnishMaxSpeed(ADR(OverVarnish), ADR(gBelt));
	rStackerMaxSpeed := StackerMaxSpeed(ADR(Stacker), ADR(gBelt));

	gLine.Parameters.Hw.rMaxSpeed := MIN(rFeederMaxSpeed, rPrimerMaxSpeed, rSarmMaxSpeed, rDryerMaxSpeed, rOvervarnishMaxSpeed, rStackerMaxSpeed);

	gLine.Parameters.Hw.rMaxSpeed := MIN(rLineMaxSpeed, gLine.Parameters.Hw.rMaxSpeed);

END_ACTION

ACTION DefineLineFeaturesAllowed:

	gLine.Parameters.Hw.xDoubleLineAllowed := 	(Feeder.Parameters.Hw.xDoubleLineAllowed OR NOT Feeder.ParSw.xEnabled) AND
												(Primer.Parameters.Hw.xDoubleLineAllowed OR NOT Primer.ParSw.xEnabled) AND
												(Sarm.Parameters.Hw.xDoubleLineAllowed OR NOT Sarm.ParSw.xEnabled) AND
												(Dryer.Parameters.Hw.xDoubleLineAllowed OR NOT Dryer.ParSw.xEnabled) AND
												(OverVarnish.Parameters.Hw.xDoubleLineAllowed OR NOT OverVarnish.ParSw.xEnabled) AND
												(Stacker.Parameters.Hw.xDoubleLineAllowed OR NOT Stacker.ParSw.xEnabled);

END_ACTION
```

#### LineInputs.st
```iecst
ACTION LineInputs:

	tonLineNotPowered.IN:= NOT Line.Inputs.xPrinterPowered; //Line.Inputs.UPSs[1].LoadOnBattery OR Line.Inputs.UPSs[2].LoadOnBattery;
	tonLineNotPowered.PT:=T#20s;
	tonLineNotPowered();
	xLinePowered := NOT tonLineNotPowered.Q;

	//Start order
	tonLineStartButton(IN:=gMachine.In.Buttons.xStart, PT:=T#1s);

END_ACTION
```

#### LineOutputs.st
```iecst
ACTION LineOutputs:

	//Ancillaries present inputs
	Feeder.Inputs.xFeederPresent := Line.Outputs.ExternalDevices[0].xClose;
	Primer.Inputs.xPrimerPresent := Line.Outputs.ExternalDevices[1].xClose;
	OverVarnish.Inputs.xOPVPresent := Line.Outputs.ExternalDevices[10].xClose;
	Stacker.Inputs.xStackerPresent := Line.Outputs.ExternalDevices[6].xClose;
	Sarm.Inputs.xSarmPresent := Line.Outputs.ExternalDevices[11].xClose;

	//DryerRemoteData

	//Commands
	DryerData.Commands.xPrepareToDry := Dryer.Outputs.xPrepareToDry;
	DryerData.Commands.xStartDrying := Dryer.Outputs.xStartDrying;
	DryerData.Commands.xPrepareToEmptyBelt := Dryer.Outputs.xPrepareToEmptyBelt;

	DryerData.Parameters.xEnableNir := Dryer.ParSw.xEnableNIR;
	DryerData.Parameters.xEnableArcLamp := Dryer.ParSw.xEnableArcLamp;
	DryerData.Parameters.xEnableDDC := Dryer.ParSw.xEnableDDC;

	//Parameters
	DryerData.Parameters.rBeltSpeedSetPoint := Dryer.Parameters.rSpeedSetPoint;
	DryerData.Parameters.Media.rThickness := Dryer.Parameters.rMediaThickness;
	DryerData.Parameters.Media.rWidth := Dryer.Parameters.rMediaWidth;
	DryerData.Parameters.Media.rLength := Dryer.Parameters.rMediaLength;
	DryerData.Parameters.Media.rCrossOffset := gMachine.parSw.Media.rOffsetRegisterL1;

	DryerData.Parameters.Media.rDocWidth := Dryer.Parameters.rDocumentWidth;
	DryerData.Parameters.Media.rDocLength := Dryer.Parameters.rDocumentLength;
	DryerData.Parameters.Media.rDocCrossOffset := Dryer.Parameters.rDocumentOffsetL1; //NOZDRYER-467
	//DryerData.Parameters.Document.rOffsetL2 := Dryer.Parameters.rDocumentOffsetL2; //NOZDRYER-467
	DryerData.Parameters.xDoubleLine := Dryer.Parameters.xDoubleLine;
	DryerData.Parameters.xLineEmptyingBelt := Line.StatusSummary.xEmptyingBelts;
	DryerData.Parameters.xPrinterBeltRuning := Belt.states.xRuningBelt;
	DryerData.Parameters.rSubstratePowerReduction := Dryer.ParSw.rSubstratePowerReduction;

	//Signals
	DryerData.Signals.xMediaPresent := ThickCtrl.status.MediaPosition.xMediaAtPrinterExit; //Dryer.Inputs.xMediaPresent
	//DryerData.Signals.xBreakerOKBlowerInput := Line_X20DIF371_003.DInput[15];  //Mapping done directly in plc card assignation
	//DryerData.Signals.xBreakerOKBlowerOutput := Line_X20DIF371_003.DInput[16];  //Mapping done directly in plc card assignation

	DryerData.Signals.Safety.xMovementsEnabled := SafetyController.Outputs.xEnableDryer1; // AND SafetyController.Outputs.xEnableDryer2;
	DryerData.Signals.Safety.xRemoteEStopOK := NOT SafetyController.Alarms.xCriticalAlarm;
	DryerData.Signals.Safety.xEStopFrontOK := SafetyController.Inputs.xDryerFrontsideEstop;
	DryerData.Signals.Safety.xEStopRearOK := SafetyController.Inputs.xDryerBacksideEstop;
	DryerData.Signals.Safety.xClosedFrontInput := SafetyController.Inputs.xDryerFrontDoorSwitch1;
	DryerData.Signals.Safety.xClosedFrontOutput := SafetyController.Inputs.xDryerFrontDoorSwitch2;
	DryerData.Signals.Safety.xClosedRearInput := SafetyController.Inputs.xDryerBackDoorSwitch1;
	DryerData.Signals.Safety.xClosedRearOutput := SafetyController.Inputs.xDryerBackDoorSwitch2;

	IF EDGENEG(ThickCtrl.parameters.xBlockInProperPrintingPosition) AND (Line.Status=LINE_PRINTING) THEN
		Line.Outputs.Sw.iTimesBlockAtSafePosition := Line.Outputs.Sw.iTimesBlockAtSafePosition + 1;
	ELSIF Line.Status=LINE_STOPPED THEN
		Line.Outputs.Sw.iTimesBlockAtSafePosition := 0;
	END_IF

	//DELOREAN-830: To ask sw to execute a cleaning command when curing has been active when block is at safe position
	xCuringSystemStarted := CuringSystemsStarted(ADR(CuringLed[1])) OR CuringSystemsStarted(ADR(CuringLed[2]));
	IF NOT ThickCtrl.parameters.xBlockInProperPrintingPosition AND xCuringSystemStarted THEN
		xToCleanAfterBlockAtSafePosition := TRUE;
	END_IF

	//DELOREAN-830: Request SW to execute a cleaning
	//To active this output just when line is receptive to "Line.Commands.Clean"
	Line.Outputs.Sw.xCleanOrderRequestToSw := xToCleanAfterBlockAtSafePosition AND (Line.Status=LINE_IDLE);
	IF Line.StatusSummary.xCleaning OR
		EDGEPOS(Line.StatusSummary.xPrinting) OR
		EDGEPOS(Line.StatusSummary.xEmptyingBelts) THEN

		xToCleanAfterBlockAtSafePosition:=FALSE;
	END_IF

	Line.Outputs.Sw.xPrintOrderRequestToSw:=xLineRequestToPrintToSw;

END_ACTION
```

#### PreparingPrint.st
```iecst
ACTION PreparingPrint:

	IF xStatusChanged THEN
		iLineStatus:=300;
	END_IF

	CASE iLineStatus OF

		300:
			Stacker.Commands.xPrepare:=TRUE;
			//[RGP] Giving this order just when preparing to print. So media widht must not change while in printing position when EHD is active. Sw must secure that
			//The workflow would be: unload job, line goes to pause, bars go up a little bit over metal bands, then when going to print again, this order will be
			//activated again and ehd system will be adjusted to new media parameters.
			EdgeHoldDown.orders.xAdjustToMedia := TRUE;

			xStackerReady := StackerReady(ADR(Stacker));
			IF xStackerReady THEN
				Stacker.Commands.xStart:=TRUE;
				OverVarnish.Commands.xPrepare:=TRUE;
				iLineStatus:=iLineStatus+1;
			END_IF

		301:
			xEhdAdjusted := EhdAdjusted(ADR(EdgeHoldDown));
			IF xEhdAdjusted THEN
				EdgeHoldDown.orders.xAdjustToMedia := FALSE;
				Machine.commandsSw.xToNormal_GI := TRUE;
				iLineStatus:=iLineStatus+1;
			END_IF

		302:
			IF Machine.St.AutoMode.xProduction AND NOT gOverVarnish.ParSw.xEnablePriming THEN
				Machine.commandsSw.xToNormal_GI := FALSE; //TOREVIEW: This should be an internal command, not something coming from Comms
				Machine.commands.xAllToPrint:=TRUE;
				iLineStatus:=iLineStatus+1;
			ELSIF Machine.St.AutoMode.xProduction AND gOverVarnish.ParSw.xEnablePriming THEN
				iLineStatus:=iLineStatus+1;
			END_IF

		303:
			xOverVarnishReady := OpvReady(ADR(OverVarnish));
			IF xOverVarnishReady THEN
				OverVarnish.Commands.xStart := TRUE;
				IF Dryer.ParSw.xEnableNIR THEN
					Dryer.Commands.xPrepare:=TRUE;
				ELSE
					Dryer.Commands.xStartTransport:=TRUE;
				END_IF
				IF Machine.St.AutoMode.xProduction AND gOverVarnish.ParSw.xEnablePriming THEN
					Machine.commandsSw.xToNormal_GI := FALSE; //TOREVIEW: This should be an internal command, not something coming from Comms
					Machine.commands.xAllToPrint:=TRUE;
				END_IF
				iLineStatus:=iLineStatus+1;
			END_IF

		304:
			xBarsInPrintingPosition := BarPositionReady(ADR(Machine));
			//DELOREAN-1670: To check feeder ready in same step where Prepare order is being activated
			IF xBarsInPrintingPosition THEN
				iLineStatus:=iLineStatus+1;
			END_IF

		305:
			xOverVarnishReady := OpvReady(ADR(OverVarnish));
			xOverVarnishStarted := OpvStarted(ADR(OverVarnish));
			xDryerReady := DryerReady(ADR(Dryer));
			xStackerReady := StackerReady(ADR(Stacker));
			IF xDryerReady AND (xOverVarnishReady OR xOverVarnishStarted) AND xStackerReady THEN
				xLineReady:=TRUE;
			END_IF

	END_CASE

END_ACTION
```

#### StartingPrinting.st
```iecst
ACTION StartingPrinting:

	IF xStatusChanged THEN
		iLineStatus:=310;
	END_IF

	CASE iLineStatus OF
		310:
			Dryer.Commands.xStart:=TRUE;
			iLineStatus:=iLineStatus+1;

		311:
			xStackerStarted:=StackerStarted(ADR(Stacker));
			xOverVarnishStarted:=OpvStarted(ADR(OverVarnish));
			xDryerStarted:=DryerStarted(ADR(Dryer));
			xJobReady := JobReady(ADR(Machine));

			xThicknessSensorReady := ThicknessSensorReady(ADR(ThickCtrl));
			IF xThicknessSensorReady AND xDryerStarted AND xOverVarnishStarted AND xStackerStarted THEN
				//[RGP] To avoid to start printer's belt before job is loaded. This occurs when there is no feeder and user prints samples by entering boards from printer's entry
				IF Feeder.ParSw.xEnabled OR (NOT Feeder.ParSw.xEnabled AND xJobReady) THEN
					gMachine.commands.xRunBelt:=TRUE;
				END_IF
				iLineStatus:=iLineStatus+1;
			END_IF

		312:
			xPrinterBeltStarted:= PrinterBeltStarted(ADR(Belt));
			xCuringSystemReady := CuringSystemsReady(ADR(CuringLed[1])) AND CuringSystemsReady(ADR(CuringLed[2]));
			xJobReady := JobReady(ADR(Machine));

			IF xPrinterBeltStarted AND xCuringSystemReady AND xJobReady THEN
				Sarm.Commands.xStart := TRUE;
				Primer.Commands.xPrepare:=TRUE;
				iLineStatus:=iLineStatus+1;
			END_IF

		313:
			xSarmReady := SarmReady(ADR(Sarm));
			xSarmStarted:=SarmStarted(ADR(Sarm));
			xPrimerReady := PrimerReady(ADR(Primer));
			IF xPrimerReady AND (xSarmReady OR xSarmStarted) THEN
				Primer.Commands.xStart := TRUE;
				iLineStatus:=iLineStatus+1;
			END_IF
		314:
			xPrimerStarted:=PrimerStarted(ADR(Primer));
			xSarmStarted:=SarmStarted(ADR(Sarm));
			IF xPrimerStarted AND xSarmStarted THEN
				Feeder.Commands.xPrepare:=TRUE;
				iLineStatus:=iLineStatus+1;
			END_IF

		315:
			IF NOT xLineToPause THEN
				xFeederReady := FeederReady(ADR(Feeder));
				IF xFeederReady THEN
					Feeder.Commands.xStart:=TRUE;
					iLineStatus:=iLineStatus+1;
				END_IF
			ELSE
				xLineReady:=TRUE;
			END_IF

		316:
			IF NOT xLineToPause THEN
				xFeederStarted:=FeederStarted(ADR(Feeder));
				IF xFeederStarted THEN
					xLineReady:=TRUE;
				END_IF
			ELSE
				xLineReady:=TRUE;
			END_IF

	END_CASE

END_ACTION
```

#### PreparingCleaningPH.st
```iecst
ACTION PreparingCleaningPH:

	IF xStatusChanged THEN
		iLineStatus:=400;
	END_IF

	CASE iLineStatus OF
		400:
			gMachine.commands.xClean:=TRUE;
			xLineReady:=TRUE;

	END_CASE

END_ACTION
```

#### StartingCleaningPH.st
```iecst
ACTION StartingCleaningPH:

	IF xStatusChanged THEN
		iLineStatus:=410;
	END_IF

	CASE iLineStatus OF
		410:
			xBarsInCleaningPosition := BarPositionCleaning(ADR(Machine));
			IF xBarsInCleaningPosition THEN
				gMachine.commands.xClean:=FALSE;
				iLineStatus:=0;
				xLineReady:=TRUE;
			END_IF
	END_CASE

END_ACTION
```

#### StartingCleaningBelt.st
```iecst
ACTION StartingCleaningBelt:

	IF xStatusChanged THEN
		iLineStatus:=710;
	END_IF

	CASE iLineStatus OF
		710:
			IF BeltClean.Status.xCleaning OR gBeltClean.Status.State = BCLEAN_FAULT THEN
				gMachine.commands.CleanBelt.xStart := FALSE;
				xCleanBeltToBeExecuted := FALSE;
				xLineReady:=TRUE;
			END_IF
	END_CASE

END_ACTION
```

#### Stopping.st
```iecst
ACTION Stopping:

	IF xStatusChanged THEN
		iLineStatus:=650;
	END_IF

	CASE iLineStatus OF
		650:
			StopAllLineDevices;
			iLineStatus:=iLineStatus+1;

		651:
			xFeederStopped:=FeederStopped(ADR(Feeder));
			xPrimerStopped:=PrimerStopped(ADR(Primer));
			xSarmStopped := SarmStopped(ADR(Sarm));
			xDryerStopped:=DryerStopped(ADR(Dryer));
			xOverVarnishStopped:=OpvStopped(ADR(OverVarnish));
			xStackerStopped:=StackerStopped(ADR(Stacker));
			xEhdStopped := EhdStopped(ADR(EdgeHoldDown));
			IF xFeederStopped AND xPrimerStopped AND xDryerStopped AND xStackerStopped AND xOverVarnishStopped AND xEhdStopped AND xSarmStopped THEN
				xLineReady:=TRUE;
			END_IF

	END_CASE

END_ACTION

ACTION StopAllLineDevices:
	Feeder.Commands.xStop:=TRUE;
	Primer.Commands.xStop:=TRUE;
	Sarm.Commands.xStop:=TRUE;
	Dryer.Commands.xStop:=TRUE;
	OverVarnish.Commands.xStop:=TRUE;
	Stacker.Commands.xStop:=TRUE;
	gMachine.commands.xStop:=TRUE;
	gMachine.commands.xClean:=FALSE;
	gMachine.commands.CleanBelt.xStart := FALSE;
	gMachine.St.xAbortJobRequest:=TRUE;
	gMachine.commands.xRunBelt:=FALSE; //This shouldnt be required, Why stop command does not stop the belt?
	EdgeHoldDown.orders.xAdjustToMedia:=FALSE;
	EdgeHoldDown.orders.xResetPosition:=FALSE;
	EdgeHoldDown.commands.xStop:=TRUE;
	StopCuringSystems;
	StopBlowers;
END_ACTION
```

#### LightTowerManagement.st - Alarms sound
```iecst
ACTION LightTower:

	IF Line.Status<>LINE_NOT_INITIALIZED THEN
		// White: Line in automatic mode
		Line.Outputs.xWhiteLight:= gMachine.St.Mode.xAuto;

		// Blue: Any alarm may be reset
		Line.Outputs.xBlueLight := Line.Alarms.xResetCondition;

		// Green:
		//Light tower's green light is managed by safety controller physical output
		//Management done below is not related to light tower so green light button on HMI panel.
		IF (Line.Status=LINE_IDLE AND gMachine.parSw.UI.xStartPrintButtonActive AND xNoAlarmsActive) OR (gMachine.St.xRobotReadyToPrint AND Line.Status=LINE_PAUSED) THEN
			Line.Outputs.xGreenLight := gPLC.xBlk_500ms;
		ELSIF Belt.states.xRuningBelt THEN
			Line.Outputs.xGreenLight := TRUE;
		ELSE
			Line.Outputs.xGreenLight := FALSE;
		END_IF

		// Red: Safety related alarm
		Line.Outputs.xRedLight := SafetyController.Alarms.xCriticalAlarm;

		// Yellow Blinking: warning
		IF (Line.Alarms.xCriticalAlarm OR Line.Alarms.xStopAlarm) THEN
			Line.Outputs.xYellowLight := gPLC.xBlk_1s;
		// Yellow Solid: warning
		ELSIF Line.Alarms.xWarningAlarm THEN
			Line.Outputs.xYellowLight := TRUE;
		ELSE
			Line.Outputs.xYellowLight := FALSE;
		END_IF

		iIndexLights := 1;
		iIndexLightsAux := iNumberOfLights;

	ELSE
		InitializingLights;

	END_IF

END_ACTION

ACTION SoundLightTower:
	// Acoustic advise
	//
	// AutoReseteable Alarms sound management
	//arCriticalMachine (xAlarm:= gMachine.AlSummary.xAlarmCritical, xSilence:=gMachine.AutoCmd.xMuteAlarms);
	arCriticalDryer (xAlarm:= Dryer.Alarms.xCriticalAlarm, xSilence:=gMachine.AutoCmd.xMuteAlarms);
	arCriticalStacker (xAlarm:= Stacker.Alarms.xCriticalAlarm, xSilence:=gMachine.AutoCmd.xMuteAlarms);
	arCriticalSafetyFeeder (xAlarm:= SafetyController.Alarms.xAlrFeeder, xSilence:=gMachine.AutoCmd.xMuteAlarms);
	arCriticalSafetyPrimer (xAlarm:= SafetyController.Alarms.xAlrPrimer, xSilence:=gMachine.AutoCmd.xMuteAlarms);
	arCriticalSafetyDryer (xAlarm:= SafetyController.Alarms.xAlrDryer, xSilence:=gMachine.AutoCmd.xMuteAlarms);
	arCriticalSafetyOverVarnish (xAlarm:= SafetyController.Alarms.xAlrOverVarnish, xSilence:=gMachine.AutoCmd.xMuteAlarms);
	arCriticalSafetyStacker (xAlarm:= SafetyController.Alarms.xAlrStacker, xSilence:=gMachine.AutoCmd.xMuteAlarms);
	arCriticalSafetyDoorLock (xAlarm:= SafetyController.Alarms.xAlrPrinterDoorLock, xSilence:=gMachine.AutoCmd.xMuteAlarms);
	arCriticalSafetyLightCurtain (xAlarm:= (SafetyController.Alarms.xAlrPrinterLightCurtain AND NOT gMachine.St.Mode.xZero), xSilence:=gMachine.AutoCmd.xMuteAlarms);
	arCriticalMachineNoPowered (xAlarm:= Line.Alarms.xAlrPrinterNoPowered, xSilence:=gMachine.AutoCmd.xMuteAlarms);
	arCriticalOvervoltage (xAlarm:= Line.Alarms.xAlrOvervoltage, xSilence:=gMachine.AutoCmd.xMuteAlarms);
	arCritical24vdcStartSeqNoPowered (xAlarm:= Line.Alarms.xAlr24VdcStartSeqNoPowered, xSilence:=gMachine.AutoCmd.xMuteAlarms);
	//arCriticalStopButton (xAlarm:= gMachine.In.Buttons.xStop, xSilence:=gMachine.AutoCmd.xMuteAlarms); //To not sound due to issue: NOZOMITWO-1027
	arCriticalSafetySarm (xAlarm:= SafetyController.Alarms.xAlrSarm, xSilence:=gMachine.AutoCmd.xMuteAlarms);

	arStop	(xAlarm:= Line.Alarms.xStopAlarm, xSilence:=gMachine.AutoCmd.xMuteAlarms);

	tp_RejectSound.IN:=ThickCtrl.Outputs.xReject;
	tp_RejectSound.PT:=T#1S;
	tp_RejectSound();

	iReasonSound.0 := arCriticalMachine.xAlarmSound;
	iReasonSound.1 := arCriticalDryer.xAlarmSound;
	iReasonSound.2 := arCriticalStacker.xAlarmSound;
	iReasonSound.3 := arCriticalSafetyFeeder.xAlarmSound;
	iReasonSound.4 := arCriticalSafetyPrimer.xAlarmSound;
	iReasonSound.5 := arCriticalSafetyDryer.xAlarmSound;
	iReasonSound.6 := arCriticalSafetyStacker.xAlarmSound;
	iReasonSound.7 := arCriticalSafetyDoorLock.xAlarmSound;
	iReasonSound.8 := arCriticalSafetyLightCurtain.xAlarmSound;
	iReasonSound.9 := arCriticalMachineNoPowered.xAlarmSound;
	iReasonSound.10 := arCriticalOvervoltage.xAlarmSound;
	iReasonSound.11 := arCritical24vdcStartSeqNoPowered.xAlarmSound;
	iReasonSound.12 := arStop.xAlarmSound;
	iReasonSound.13 := tp_RejectSound.Q;
	iReasonSound.14 := arCriticalSafetySarm.xAlarmSound;

	// Alarm sound output
	Line.Alarms.xAlarmSound := iReasonSound > 0;
	Line.Outputs.xSound :=  iReasonSound > 0;

END_ACTION

ACTION InitializingLights:
		IF iIndexLights<iNumberOfLights THEN
			IF iIndexLightsAux>=iIndexLights THEN
				IF EDGEPOS(gPLC.xBlk_200ms) THEN
					FOR iLights:=iIndexLights+1 TO iNumberOfLights DO
						gArrayLights[iLights]:= FALSE;
					END_FOR
					gArrayLights[iIndexLightsAux]:= TRUE;
					iIndexLightsAux := MAX(0, iIndexLightsAux - 1);
				END_IF
			ELSE
				iIndexLights := iIndexLights + 1;
				iIndexLightsAux := iNumberOfLights;
			END_IF

		ELSIF iRepeatTimes<=5 THEN
			IF EDGEPOS(gPLC.xBlk_500ms) THEN
				iRepeatTimes:=iRepeatTimes+1;
				FOR iLights:=1 TO iNumberOfLights DO
					gArrayLights[iLights]:= FALSE;
				END_FOR

			ELSIF EDGENEG(gPLC.xBlk_500ms) THEN
				FOR iLights:=1 TO iNumberOfLights DO
					gArrayLights[iLights]:= TRUE;
				END_FOR
			END_IF

		ELSE
			iIndexLights := 1;
			iRepeatTimes := 1;
		END_IF

		//Assigning to each color
		Line.Outputs.xWhiteLight 	:= gArrayLights[1];
		Line.Outputs.xBlueLight 	:= gArrayLights[2];
		Line.Outputs.xGreenLight 	:= gArrayLights[3];
		Line.Outputs.xYellowLight 	:= gArrayLights[4];
		Line.Outputs.xRedLight 		:= gArrayLights[5];
END_ACTION
```

#### PowerOffLineDevices.st
```iecst
ACTION PowerOffLineDevices:

	IF xStatusChanged THEN
		iLineStatus:=100;
		iIndexPower:=0;
		xLinePoweredOFF:=FALSE;
	END_IF

	CASE iLineStatus OF
		100:
			ton_DelayPowerOff.IN := TRUE;
			ton_DelayPowerOff.PT := t#3s;
			ton_DelayPowerOff();

			IF iIndexPower<=Line.Parameters.iNumExternalDevices THEN

				IF Line.Parameters.ExternalDevices[iIndexPower].xIsEngine THEN
					Line.Outputs.ExternalDevices[iIndexPower].xClose:=FALSE;

					IF ton_DelayPowerOff.Q THEN
						//Reset the output
						Line.Outputs.ExternalDevices[iIndexPower].xOpen:=FALSE;

						//Reset timer
						ResetPowerOffTimerAndNext;
					END_IF

				ELSE
					//Reset the outputs
					Line.Outputs.ExternalDevices[iIndexPower].xOpen:=FALSE;
					Line.Outputs.ExternalDevices[iIndexPower].xClose:=FALSE;

					ResetPowerOffTimerAndNext;
				END_IF

			ELSE
				iLineStatus:=iLineStatus+1;
			END_IF

		101:
			xLinePoweredOFF:=TRUE;

	END_CASE

END_ACTION

ACTION ResetPowerOffTimerAndNext:

	//Reset timer
	ton_DelayPowerOff(IN:=FALSE);
	iIndexPower:=iIndexPower+1;

END_ACTION
```

#### EventLog.st
```iecst
ACTION LogWarningAlarm:

	stWarningAlarmsLog.Source := ELOG_TYPE_GENERAL;
	stWarningAlarmsLog.Severity:= ELOG_SEVERITY_INFO;
	stWarningAlarmsLog.Facility:= 0;
	stWarningAlarmsLog.ErrorCode:=0;

	stWarningAlarmsLog.Text := 'Line.LogWarningAlarm';

	IF iReasonWarning.0 THEN stWarningAlarmsLog.Text := 'gMachine.AlSummary.xAnyWarning';
	ELSIF iReasonWarning.1 THEN	stWarningAlarmsLog.Text := 'Feeder.Alarms.xWarningAlarm';
	ELSIF iReasonWarning.2 THEN	stWarningAlarmsLog.Text := 'Primer.Alarms.xWarningAlarm';
	ELSIF iReasonWarning.3 THEN stWarningAlarmsLog.Text := 'Dryer.Alarms.xWarningAlarm';
	ELSIF iReasonWarning.4 THEN stWarningAlarmsLog.Text := 'Stacker.Alarms.xWarningAlarm';
	ELSIF iReasonWarning.5 THEN stWarningAlarmsLog.Text := 'SafetyController.Alarms.xWarningAlarm';
	ELSIF iReasonWarning.6 THEN stWarningAlarmsLog.Text := 'Sarm.Alarms.xWarningAlarm';
	END_IF

	gEventLogLoader(EventData := ADR(stWarningAlarmsLog));

END_ACTION

ACTION LogStopAlarm:

	stStopAlarmsLog.Source := ELOG_TYPE_GENERAL;
	stStopAlarmsLog.Severity:= ELOG_SEVERITY_INFO;
	stStopAlarmsLog.Facility:= 0;
	stStopAlarmsLog.ErrorCode:=0;

	stStopAlarmsLog.Text := 'Line.LogStopAlarm';

	IF iReasonStop.0 THEN stStopAlarmsLog.Text := 'gMachine.AlSummary.xAlarmStop';
	ELSIF iReasonStop.1 THEN stStopAlarmsLog.Text := 'Primer.Alarms.xCriticalAlarm';
	ELSIF iReasonStop.2 THEN stStopAlarmsLog.Text := 'Line.Commands.Stop';
	ELSIF iReasonStop.3 THEN stStopAlarmsLog.Text := 'CuringLed[1].AlSummary.xAlarmStop';
	ELSIF iReasonStop.4 THEN stStopAlarmsLog.Text := 'CuringLed[2].AlSummary.xAlarmStop';
	ELSIF iReasonStop.5 THEN stStopAlarmsLog.Text := 'EdgeHoldDown.AlSummary.xAlarmStop';
	ELSIF iReasonStop.6 THEN stStopAlarmsLog.Text := 'Sarm.Alarms.xCriticalAlarm';
	END_IF

	gEventLogLoader(EventData := ADR(stStopAlarmsLog));

END_ACTION

ACTION LogCriticalAlarm:

	stCriticalAlarmsLog.Source := ELOG_TYPE_GENERAL;
	stCriticalAlarmsLog.Severity:= ELOG_SEVERITY_ERROR;
	stCriticalAlarmsLog.Facility:=0;
	stCriticalAlarmsLog.ErrorCode:=0;

	stCriticalAlarmsLog.Text := 'Line.LogCriticalAlarm';

	IF iReasonCritical.0 THEN stCriticalAlarmsLog.Text := 'gMachine.AlSummary.xAlarmCritical';
	ELSIF iReasonCritical.1 THEN stCriticalAlarmsLog.Text := 'Dryer.Alarms.xCriticalAlarm';
	ELSIF iReasonCritical.2 THEN stCriticalAlarmsLog.Text := 'Stacker.Alarms.xCriticalAlarm';
	ELSIF iReasonCritical.3 THEN stCriticalAlarmsLog.Text := 'SafetyController.Alarms.xCriticalAlarm';
	ELSIF iReasonCritical.4 THEN stCriticalAlarmsLog.Text := 'Line.Alarms.xAlrPrinterNoPowered';
	ELSIF iReasonCritical.5 THEN stCriticalAlarmsLog.Text := 'Line.Alarms.xAlr400VacNok';
	ELSIF iReasonCritical.6 THEN stCriticalAlarmsLog.Text := 'Line.Alarms.xAlr24VdcStartSeqNoPowered';
	ELSIF iReasonCritical.7 THEN stCriticalAlarmsLog.Text := 'gMachine.In.Buttons.xStop';
	ELSIF iReasonCritical.8 THEN stCriticalAlarmsLog.Text := 'OverVarnish.Alarms.xCriticalAlarm';
	ELSIF iReasonCritical.9 THEN stCriticalAlarmsLog.Text := 'CuringLed[1].AlSummary.xAlarmCritical';
	ELSIF iReasonCritical.10 THEN stCriticalAlarmsLog.Text := 'CuringLed[2].AlSummary.xAlarmCritical';
	ELSIF iReasonCritical.11 THEN stCriticalAlarmsLog.Text := 'EdgeHoldDown.AlSummary.xAlarmCritical';
	END_IF

	gEventLogLoader(EventData := ADR(stCriticalAlarmsLog));

END_ACTION

ACTION LogPrintCommand:

	stPrintCommandLog.Source := ELOG_TYPE_GENERAL;
	stPrintCommandLog.Severity:= ELOG_SEVERITY_INFO;
	stPrintCommandLog.Facility:= 0;
	stPrintCommandLog.ErrorCode:=0;

	stPrintCommandLog.Text := 'Line.LogPrintCommand';

	gEventLogLoader(EventData := ADR(stPrintCommandLog));

END_ACTION

ACTION LogPauseCommand:

	stPauseCommandLog.Source := ELOG_TYPE_GENERAL;
	stPauseCommandLog.Severity:= ELOG_SEVERITY_INFO;
	stPauseCommandLog.Facility:= 0;
	stPauseCommandLog.ErrorCode:=0;

	stPauseCommandLog.Text := 'Line.LogPauseCommand';

	gEventLogLoader(EventData := ADR(stPauseCommandLog));

END_ACTION

ACTION LogCleanCommand:

	stCleanCommandLog.Source := ELOG_TYPE_GENERAL;
	stCleanCommandLog.Severity:= ELOG_SEVERITY_INFO;
	stCleanCommandLog.Facility:= 0;
	stCleanCommandLog.ErrorCode:=0;

	stCleanCommandLog.Text := 'Line.LogCleanCommand';

	gEventLogLoader(EventData := ADR(stCleanCommandLog));

END_ACTION

ACTION LogEmptyBeltCommand:

	stEmptyBeltCommandLog.Source := ELOG_TYPE_GENERAL;
	stEmptyBeltCommandLog.Severity:= ELOG_SEVERITY_INFO;
	stEmptyBeltCommandLog.Facility:= 0;
	stEmptyBeltCommandLog.ErrorCode:=0;

	stEmptyBeltCommandLog.Text := 'Line.LogEmptyBeltCommand';

	gEventLogLoader(EventData := ADR(stEmptyBeltCommandLog));

END_ACTION

ACTION LogStopCommand:

	stStopCommandLog.Source := ELOG_TYPE_GENERAL;
	stStopCommandLog.Severity:= ELOG_SEVERITY_INFO;
	stStopCommandLog.Facility:= 0;
	stStopCommandLog.ErrorCode:=0;

	stStopCommandLog.Text := 'Line.LogStopCommand';

	gEventLogLoader(EventData := ADR(stStopCommandLog));

END_ACTION

ACTION LogStartButton:

	stStartButtonLog.Source := ELOG_TYPE_GENERAL;
	stStartButtonLog.Severity:= ELOG_SEVERITY_INFO;
	stStartButtonLog.Facility:= 0;
	stStartButtonLog.ErrorCode:=0;

	stStartButtonLog.Text := 'Line.LogStartButton';

	gEventLogLoader(EventData := ADR(stStartButtonLog));

END_ACTION

ACTION LogStopButton:

	stStopButtonLog.Source := ELOG_TYPE_GENERAL;
	stStopButtonLog.Severity:= ELOG_SEVERITY_INFO;
	stStopButtonLog.Facility:= 0;
	stStopButtonLog.ErrorCode:=0;

	stStopButtonLog.Text := 'Line.LogStopButton';

	gEventLogLoader(EventData := ADR(stStopButtonLog));

END_ACTION

ACTION LogLineSubStatus:

	stLineSubStatusLog.Source := ELOG_TYPE_GENERAL;
	stLineSubStatusLog.Severity:= ELOG_SEVERITY_INFO;
	stLineSubStatusLog.Facility:= 0;
	stLineSubStatusLog.ErrorCode:=0;

	stLineSubStatusLog.Text := 'LogLineSubStatus = ';
	stSubStatus := INT_TO_STRING(Line.SubStatus);
	strcat(ADR(stLineSubStatusLog.Text), ADR(stSubStatus));
	//stLineSubStatusLog.Text := INT_TO_STRING(Line.SubStatus);

	gEventLogLoader(EventData := ADR(stLineSubStatusLog));

END_ACTION

ACTION LogLineSwStatus:

	stLineStatusSwLog.Source := ELOG_TYPE_GENERAL;
	stLineStatusSwLog.Severity:= ELOG_SEVERITY_INFO;
	stLineStatusSwLog.Facility:= 0;
	stLineStatusSwLog.ErrorCode:=0;

	stLineStatusSwLog.Text := 'LogLineSwStatus = ';
	stStatusSw := INT_TO_STRING(Line.StatusSw);
	strcat(ADR(stLineStatusSwLog.Text), ADR(stStatusSw));
	//stLineStatusSwLog.Text := INT_TO_STRING(Line.StatusSw);

	gEventLogLoader(EventData := ADR(stLineStatusSwLog));

END_ACTION
```

#### SystemsPaused.st
```iecst
(* TODO: Add your comment here *)

FUNCTION DryerPaused
	DryerPaused:=NOT Dryer.ParSw.xEnabled OR NOT Dryer.Parameters.xInstalled OR Dryer.Status.CtrlStatus=DRYERCTRL_PAUSED OR Dryer.Status.CtrlStatus=DRYERCTRL_MOVING;
END_FUNCTION

FUNCTION PrimerPaused
	PrimerPaused:=NOT Primer.ParSw.xEnabled OR NOT Primer.Parameters.xInstalled OR Primer.Status.CtrlStatus=PRIMERCTRL_PAUSED;
END_FUNCTION

FUNCTION FeederPaused
	FeederPaused:=NOT Feeder.ParSw.xEnabled OR NOT Feeder.Parameters.xInstalled OR Feeder.Status.CtrlStatus=FEEDERCTRL_PAUSED;
END_FUNCTION

FUNCTION OpvPaused
	OpvPaused:=NOT OverVarnish.ParSw.xEnabled OR NOT OverVarnish.Parameters.xInstalled OR OverVarnish.Status.CtrlStatus=OPVCTRL_PAUSED;
END_FUNCTION

FUNCTION SarmPaused
	SarmPaused:=NOT Sarm.ParSw.xEnabled OR NOT Sarm.Parameters.xInstalled OR Sarm.Status.CtrlStatus=SARMCTRL_PAUSED;
END_FUNCTION
```

#### SystemsEmptied.st
```iecst
(* TODO: Add your comment here *)

FUNCTION FeederEmptied
	FeederEmptied:=NOT Feeder.ParSw.xEnabled OR NOT Feeder.Parameters.xInstalled OR Feeder.Status.CtrlStatus<>FEEDERCTRL_FEEDING;
END_FUNCTION

FUNCTION PrimerEmptied
	PrimerEmptied:=NOT Primer.ParSw.xEnabled OR NOT Primer.Parameters.xInstalled OR Primer.Status.xBeltEmpty;
END_FUNCTION

FUNCTION PrinterEmptied
	PrinterEmptied:= ThickCtrl.status.Belt.xBeltEmpty;
END_FUNCTION

FUNCTION DryerEmptied
	DryerEmptied:=NOT Dryer.ParSw.xEnabled OR NOT Dryer.Parameters.xInstalled OR Dryer.Status.xBeltEmpty;
END_FUNCTION

FUNCTION OpvEmptied
	OpvEmptied:=NOT OverVarnish.ParSw.xEnabled OR NOT OverVarnish.Parameters.xInstalled OR OverVarnish.Status.xBeltEmpty;
END_FUNCTION

FUNCTION StackerEmptied
	StackerEmptied:=NOT Stacker.ParSw.xEnabled OR NOT Stacker.Parameters.xInstalled OR (Stacker.Inputs.Comms.xBeltsEmpty AND NOT Stacker.Inputs.Comms.xStackExit) OR Stacker.Status.xBeltEmpty;
END_FUNCTION

FUNCTION SarmEmptied
	SarmEmptied:=NOT Sarm.ParSw.xEnabled OR NOT Sarm.Parameters.xInstalled OR Sarm.Status.xBeltEmpty;
END_FUNCTION
```

#### SystemsStopped.st
```iecst
(* TODO: Add your comment here *)
FUNCTION FeederStopped
	FeederStopped:=NOT Feeder.ParSw.xEnabled OR NOT Feeder.Parameters.xInstalled OR Feeder.Status.CtrlStatus=FEEDERCTRL_STOPPED;
END_FUNCTION

FUNCTION PrimerStopped
	PrimerStopped:=NOT Primer.ParSw.xEnabled OR NOT Primer.Parameters.xInstalled OR Primer.Status.CtrlStatus=PRIMERCTRL_STOPPED;
END_FUNCTION

FUNCTION SarmStopped
	SarmStopped:=NOT Sarm.ParSw.xEnabled OR NOT Sarm.Parameters.xInstalled OR Sarm.Status.CtrlStatus=SARMCTRL_STOPPED;
END_FUNCTION

FUNCTION DryerStopped
	DryerStopped:=NOT Dryer.ParSw.xEnabled OR NOT Dryer.Parameters.xInstalled OR Dryer.Status.CtrlStatus=DRYERCTRL_STOPPED;
END_FUNCTION

FUNCTION OpvStopped
	OpvStopped:=NOT OverVarnish.ParSw.xEnabled OR NOT OverVarnish.Parameters.xInstalled OR OverVarnish.Status.CtrlStatus=OPVCTRL_STOPPED;
END_FUNCTION

FUNCTION StackerStopped
	StackerStopped:=NOT Stacker.ParSw.xEnabled OR NOT Stacker.Parameters.xInstalled OR Stacker.Status.CtrlStatus=STACKERCTRL_STOPPED;
END_FUNCTION

FUNCTION FeederNotFeeding
	FeederNotFeeding:=NOT Feeder.ParSw.xEnabled OR NOT Feeder.Parameters.xInstalled OR Feeder.Status.CtrlStatus=FEEDERCTRL_PAUSED OR Feeder.Status.CtrlStatus=FEEDERCTRL_STOPPED;
END_FUNCTION

FUNCTION PrinterBeltStopped
	PrinterBeltStopped:= NOT Belt.states.xRuningBelt;
END_FUNCTION

FUNCTION EhdStopped
	EhdStopped:=NOT EdgeHoldDown.parSw.xEnable OR NOT EdgeHoldDown.parameters.xInstalled OR NOT EdgeHoldDown.status.xMoving;
END_FUNCTION
```

#### LineCtrl.var - Local variables
```iecst
VAR
	Machine : REFERENCE TO StGeneral;
	SafetyController : REFERENCE TO stSafetyController;
	Line : REFERENCE TO LineControl_typ;
	DryerData : REFERENCE TO DryerRemoteData;
	Dryer : REFERENCE TO DryerAnc_typ;
	Feeder : REFERENCE TO Feeder_typ;
	Sarm : REFERENCE TO Sarm_typ;
	Primer : REFERENCE TO Primer_typ;
	OverVarnish : REFERENCE TO Opv_typ;
	Stacker : REFERENCE TO Stacker_typ;
	ThickCtrl : REFERENCE TO stThicknessCtrl_typ;
	EdgeHoldDown : REFERENCE TO EdgeHoldDown_typ;
	CuringLed : REFERENCE TO ARRAY[0..MAX_LAST_CURING_LED] OF CuringLed_typ;
	TransVacuum : REFERENCE TO ARRAY[0..MAX_LAST_TRANS_VACUUM] OF TransVacuum_typ;
	Belt : REFERENCE TO stBelt;
	BeltClean : REFERENCE TO BeltClean_typ;
	iLineStatus : UINT;
	xThicknessSensorReady : BOOL;
	xBarsInCleaningPosition : BOOL;
	xBarsInCapPosition : BOOL;
	xJobReady : BOOL;
	xBarsInPrintingPosition : BOOL;
	xCuringSystemStarted : BOOL;
	xCuringSystemReady : BOOL;
	xDryerPaused : BOOL;
	xDryerReady : BOOL;
	xFeederPaused : BOOL;
	rDryerMaxSpeed : REAL;
	iDryerMediaLength : UINT;
	iDryerMaxMediaThickness : UINT;
	iDryerMinMediaThickness : UINT;
	iDryerMediaWidth : UINT;
	rLineMaxSpeed : REAL := 120;
	rStackerMaxSpeed : REAL;
	iStackerMediaWidth : UINT;
	iStackerMediaLength : UINT;
	iStackerMaxMediaThickness : UINT;
	iStackerMinMediaThickness : UINT;
	rPrimerMaxSpeed : REAL;
	iPrimerMediaLength : UINT;
	iPrimerMaxMediaThickness : UINT;
	iPrimerMinMediaThickness : UINT;
	iPrimerMediaWidth : UINT;
	rOvervarnishMaxSpeed : REAL;
	iOvervarnishMediaLength : UINT;
	iOvervarnishMaxMediaThickness : UINT;
	iOvervarnishMinMediaThickness : UINT;
	iOverVarnishMinMediaThickness : UINT;
	iOverVarnishMaxMediaThickness : UINT;
	iOvervarnishMediaWidth : UINT;
	rFeederMaxSpeed : REAL;
	iFeederMediaLength : UINT;
	iFeederMinMediaThickness : UINT;
	iFeederMaxMediaThickness : UINT;
	iFeederMediaWidth : UINT;
	rSarmMaxSpeed : REAL;
	iSarmMediaWidth : UINT;
	iSarmMinMediaThickness : UINT;
	iSarmMaxMediaThickness : UINT;
	iSarmMediaLength : UINT;
	xEhdStopped : BOOL;
	xEhdAdjusted : BOOL;
	xEhdReady : BOOL;
	xFeederReady : BOOL;
	xOverVarnishPaused : BOOL;
	xOverVarnishReady : BOOL;
	xPrimerPaused : BOOL;
	xSarmReady : BOOL;
	xPrimerReady : BOOL;
	xStackerPaused : BOOL;
	xStackerReady : BOOL;
	xPrinterBeltStopped : BOOL;
	xPrinterBeltStarted : BOOL;
	xDryerStarted : BOOL;
	xFeederStarted : BOOL;
	xOverVarnishStarted : BOOL;
	xSarmStopped : BOOL;
	xSarmStarted : BOOL;
	xPrimerStarted : BOOL;
	xStackerStarted : BOOL;
	iLineSubStatusPrevious : UINT;
	LineStatusPrevious : LineStatus_enum;
	xSubStatusChanged : BOOL;
	xStatusChanged : BOOL;
	xCleanToBeExecuted : BOOL;
	xCleanBeltToBeExecuted : BOOL;
	xPreviousPausing : BOOL; (*Previously line was in paused state*)
	xPreviousPrinting : BOOL; (*Previously line was in printing state*)
	xPreviousIdle : BOOL; (*Previously line was in idle state*)
	xCleanRequestToLine : BOOL;
	xCleanDone : BOOL;
	xDryerStopped : BOOL;
	xFeederStopped : BOOL;
	xFeederNotFeeding : BOOL;
	xOverVarnishStopped : BOOL;
	ton_PrimerBeltEmpty : TON;
	ton_FeederEmpty : TON;
	ton_PrinterBeltInputEmpty : TON;
	ton_SarmBeltEmpty : TON;
	xPrimerBeltEmpty : BOOL;
	xPrinterBeltInputEmpty : BOOL;
	xSarmPaused : BOOL;
	xPrimerStopped : BOOL;
	xStackerStopped : BOOL;
	xStatesToEvaluateAlarms : BOOL;
	xLineStopped : BOOL;
	xLineReady : BOOL;
	xLinePoweredOFF : BOOL;
	xLinePoweredON : BOOL;
	tBounce : TIME;
	iIndexPower : INT;
	ton_DelayPowerOff : TON := (0);
	ton_DelayPowerOn : TON := (0);
	xLinePowered : BOOL;
	iIndexHistory : USINT;
	StateHistory : ARRAY[0..iHistoryLines] OF LineStatus_enum;
END_VAR
VAR CONSTANT
	iHistoryLines : USINT := 20;
END_VAR
VAR
	iReasonResetCondition : UDINT;
	iReasonWarning : UDINT;
	iReasonStop : UDINT;
	iReasonCritical : UDINT;
	stCriticalAlarmsLog : EventLog_typ;
	stPrintCommandLog : EventLog_typ;
	stPauseCommandLog : EventLog_typ;
	stStopCommandLog : EventLog_typ;
	stCleanCommandLog : EventLog_typ;
	stEmptyBeltCommandLog : EventLog_typ;
	stStartButtonLog : EventLog_typ;
	stStopButtonLog : EventLog_typ;
	stLineSubStatusLog : EventLog_typ;
	stLineStatusSwLog : EventLog_typ;
	stStopAlarmsLog : EventLog_typ;
	stWarningAlarmsLog : EventLog_typ;
	stStatusSw : STRING[3];
	stSubStatus : STRING[3];
	iReasonSound : UDINT;
	arCriticalMachine : AutoResetSound;
	arCriticalDryer : AutoResetSound;
	arCriticalStacker : AutoResetSound;
	arCriticalMachineNoPowered : AutoResetSound;
	arCriticalOvervoltage : AutoResetSound;
	arCritical24vdcStartSeqNoPowered : AutoResetSound;
	arCriticalStopButton : AutoResetSound;
	arCriticalSafetyFeeder : AutoResetSound;
	arCriticalSafetyPrimer : AutoResetSound;
	arCriticalSafetyOverVarnish : AutoResetSound;
	arCriticalSafetyDryer : AutoResetSound;
	arCriticalSafetyDoorLock : AutoResetSound;
	arCriticalSafetyLightCurtain : AutoResetSound;
	arCriticalSafetyStacker : AutoResetSound;
	arCriticalSafetySarm : AutoResetSound;
	arCriticalSafety : AutoResetSound;
	arStop : AutoResetSound;
	ResetedLineCommands : LineControlCommands_typ;
	AlarmsReseted : LineControlAlarms_typ;
	iLastIndexPower : INT;
	xNoAlarmsActive : BOOL;
	tonLineNotPowered : TON;
	tonLineStartButton : TON;
	xLineToEmptyBelt : BOOL;
	xLineToPrint : BOOL;
	iReasonRequestLineToPrint : UINT;
	iReasonLineToEmptyBelt : UINT;
	iReasonLineToPrint : UINT;
	tonLinePauseButton : TON;
	xLineRequestToPrintToSw : BOOL; (*Start button is pressed and lines requests SW to execute printing process*)
	xLineToClean : BOOL;
	iReasonLineToClean : UINT;
	xLineToCleanBelt : BOOL;
	iReasonLineToCleanBelt : UINT;
	xLineToPause : BOOL;
	xEhdRequestToPause : BOOL;
	rEhdBarsHeighSp : REAL;
	iReasonLineToPause : UINT;
	tp_RejectSound : TOF;
	ton_HoldOnEmptyBelt : TON; (*Timer to wait some time till evaluate line devices are empty*)
	xFeederEmptied : BOOL;
	xPrimerEmptied : BOOL;
	xPrinterEmptied : BOOL;
	xDryerEmptied : BOOL;
	xOpvEmptied : BOOL;
	xStackerEmptied : BOOL;
	xSarmEmptied : BOOL;
	xRejectHeld : BOOL;
	xLineEmpty : BOOL;
	xToCleanAfterBlockAtSafePosition : BOOL;
	xHoldOnEmptyBelt : BOOL;
	iIndexCuringLed : USINT;
	iIndexTransVacuum : USINT;
	ton_StackerCleanBelts : TON;
	tiTimeToEmpty : TIME;
	tonPrimerEmpty : TON;
	xFromPause : BOOL;
	iNumberOfLights : USINT := 5;
	gArrayLights : ARRAY[0..5] OF BOOL;
	iLights : USINT := 1;
	iIndexLightsAux : USINT := 1;
	iRepeatTimes : USINT := 1;
	iIndexLights : USINT := 1;
END_VAR
```

- LineStates.graphml (not shown)

- PowerOnOff Ancillaries.docx (binary file, 2051219 bytes)
- Doc Editor. Ghostwriter.url (not shown)

### ConfigSimulators.md
```markdown
# SIMULATORS

Configuration for the different PLC Simulators

| item      | PressPLC | DryerPLC | X5PLC |
| --------- | -------- | -------- | ----- |
| OpcUa     | 4840     | 4850     | 4845  |
| WebServer | 82       | 83       |       |
| ANSL      | 11169    | 11170    |       |
| mappView  | 84       | 81       |       |
```

- B&R System Diagnostics Manager Printer.url (not shown)

- Visualization Printer.url (not shown)

- Visualization Dryer.url (not shown)

- ProgramInitializationAndConf.graphml (not shown)

### Package Logical/Printer/Config - Machine configurator

### ReadmePrinterConfigurator.txt
```
	(* From efi Cretaprint Almazora Castellon

(*
View of the machine from the Operator side

>>>>>> LeftHandMachine 					RightHandMachine <<<<<<<<
(BK_A #1 >> BK_B #2)		LOGICAL			(BK_A #2 << BK_B #1)

Vertical:	#2 									Vertical:	#3
IclaNode: 	#5									IclaNode: 	#7
IclaIndex:	#1									IclaIndex:	#2

	          ################-################
	          ################-################
	          ################-################
	          ################-################
	##########################-###########################
	##########################-###########################
	    ######################-#######################
	    ######################-#######################
	    ######################-#######################
	    ######################-#######################

	BLOCK A [1-physical]				BLOCK B [2-physical]

*)

//Determine machine direction
	// RIGHT: gMachine.parSw.xMachineDirection is 0 or FALSE
	// LEFT:  gMachine.parSw.xMachineDirection is 1 or TRUE
	gMachine.Pt.xLeftHandMachine := gMachine.parSw.xMachineDirection;
	gMachine.Pt.xRightHandMachine:= NOT gMachine.Pt.xLeftHandMachine;

	 // P4 Config : iFirstBlock :=1  and iLastBlock :=2

	*)
```

### Program Logical/Printer/Config/Initialize (IEC)

#### Initialize.st - Cyclic code
```iecst
PROGRAM _INIT

	HWInfoCpu.pName := ADR(gMachine.St.HwData.Name);
	HWInfoCpu.first := TRUE;
	HWInfoCpu.enable := TRUE;
	HWInfoCpu();
	gMachine.St.HwData.Family := HWInfoCpu.family;
	gMachine.St.HwData.xSimulation := gMachine.St.HwData.Family = FAMILY_BRAUTOMATIONRUNTIME;

	// Tranfer permanent vars when PLC is starting

	//Recover just if there is SN in the machine
	//In the first upgrade, a character can be identified as the previous PLC version. Because of that, len>=4
	IF brsstrlen(ADR(gPermanentSN)) >= 4 OR TRUE THEN
		gMachine.St.HwData.SerialNumber := gPermanentSN;

		gMachine.parSw:= gPermanentMachine;
		gBelt.parSw:= gPermanentSwBelt;
		gBlock[1].parSw:=gPermanentBlock[1];
		gBlock[2].parSw:= gPermanentBlock[2];

		gDing.State.Permanent := gPermanentAnalogSensor;

		gSimMachine.Parameters.MachineType := gPermanentSimMachinePar.MachineType;

		FOR iInksIndex:=1 TO MAX_LAST_INK DO
			gInks[iInksIndex].parSw := gPermanentInksParSw[iInksIndex];
		END_FOR

	END_IF

END_PROGRAM

PROGRAM _CYCLIC

	//Assign the ConfigurationID been executed
	projectInfo(Execute:=gMachine.Pt.ConfigNameID=0); //Just to execute if still the configuration has not been read
	IF projectInfo.Done AND NOT projectInfo.Error THEN
		IF brsstrcmp(ADR(GC_CONFIG_2BK12BAR),ADR(projectInfo.ConfigurationID))=0 THEN
			gMachine.Pt.ConfigNameID:=GC_CONFIG_2BK12BAR_ID;
			gSimMachine.Parameters.MachineType := SIM_MACHINE_REAL;

		ELSIF brsstrcmp(ADR(GC_CONFIG_1BK2BAR),ADR(projectInfo.ConfigurationID))=0 THEN
			gMachine.Pt.ConfigNameID:=GC_CONFIG_1BK2BAR_ID;
			gSimMachine.Parameters.MachineType := SIM_MACHINE_REAL;

		ELSIF brsstrcmp(ADR(GC_CONFIG_BM_1BK8BAR),ADR(projectInfo.ConfigurationID))=0 THEN
			gMachine.Pt.ConfigNameID:=GC_CONFIG_BM_1BK8BAR_ID;
			gSimMachine.Parameters.MachineType := SIM_MACHINE_REAL;

		ELSIF brsstrcmp(ADR(GC_CONFIG_1BK8BAR_NOZ2),ADR(projectInfo.ConfigurationID))=0 THEN
			gMachine.Pt.ConfigNameID:=GC_CONFIG_1BK8BAR_NOZ2_ID;
			gSimMachine.Parameters.MachineType := SIM_MACHINE_REAL;

		ELSIF brsstrcmp(ADR(GC_CONFIG_1BK7BAR_CUBE),ADR(projectInfo.ConfigurationID))=0 THEN
			gMachine.Pt.ConfigNameID:=GC_CONFIG_1BK7BAR_CUBE_ID;
			gSimMachine.Parameters.MachineType := SIM_MACHINE_REAL;

		ELSIF brsstrcmp(ADR(GC_CONFIG_1BK10BAR_MECANO),ADR(projectInfo.ConfigurationID))=0 THEN
			gMachine.Pt.ConfigNameID:=GC_CONFIG_1BK10BAR_MECANO_ID;
			gSimMachine.Parameters.MachineType := SIM_MACHINE_REAL;

		ELSIF brsstrcmp(ADR(GC_CONFIG_1BK8BAR_NOZ2_AQ),ADR(projectInfo.ConfigurationID))=0 THEN
			gMachine.Pt.ConfigNameID:=GC_CONFIG_1BK8BAR_NOZ2_AQ_ID;
			gSimMachine.Parameters.MachineType := SIM_MACHINE_REAL;

		ELSIF brsstrcmp(ADR(GC_CONFIG_SIMTEST),ADR(projectInfo.ConfigurationID))=0 THEN
			gMachine.Pt.ConfigNameID:=GC_CONFIG_SIMTEST_ID;

		ELSIF brsstrcmp(ADR(GC_CONFIG_PLCDIAGNOSIS),ADR(projectInfo.ConfigurationID))=0 THEN
			gMachine.Pt.ConfigNameID:=GC_CONFIG_PLCDIAGNOSIS_ID;
		ELSE
			gMachine.Pt.ConfigNameID:=0;
		END_IF
		strcpy(ADR(gMachine.Pt.ConfigName),ADR(projectInfo.ConfigurationID));
	END_IF

END_PROGRAM
```

#### Initialize.var
```iecst
VAR
	HWInfoCpu : HWInfo;
	projectInfo : ArProjectGetInfo;
	iInksIndex : USINT;
END_VAR
```

### Program Logical/Printer/Config/MachineConfigurator

#### AsignCommonData.st
```iecst
ACTION AsignCommonData:

	//Just writing the fixed configuration once per each 5s
	IF NOT (EDGEPOS(gPLC.xBlk_5s) OR gPLC.xFirst_Scan OR xChangedSimMachine) THEN
		RETURN;
	END_IF

	////////////////////////////////////////////////////////////
	/////GENERAL	GENERAL		GENERAL		GENERAL	////////////
	////////////////////////////////////////////////////////////
	gMachine.Pt.CT.rMaxMarginPrinting		:= 5.0;
	gMachine.Pt.CT.rDistanceThicknesToPD	:= 187.0;

	/////////////////////////////////////////////////////
	/////BELT	BELT	BELT	BELT	BELT	BELT/////
	/////////////////////////////////////////////////////

	gBelt.parameters.IndexAxis:=1;
	gBelt.parameters.rSoftDeceleration := 1000;

	// From Units measure to meters per minute
	// Issue: CRETAPRINT LEGOCRETALEGO-964
	//These parameters only may be changed while belt is stopped for safety reasons
	IF NOT gBelt.states.xRuningBelt THEN
		gBelt.parameters.DriveUnit.TransmissionType := TRANS_LINEAL_PERIMETER;
		gBelt.parameters.DriveUnit.LinealPerimeter.PulsesPerTurn := GC_UNITS_BY_REV_DRIVE;
		gBelt.parameters.DriveUnit.LinealPerimeter.GearBox := LIMIT(1, gBelt.parSw.rGearBox, gBelt.parameters.rMaxGearBox);
		gBelt.parameters.DriveUnit.LinealPerimeter.Perimeter := LIMIT(500, gBelt.parSw.rAxisLength, gBelt.parameters.rMaxAxisLength);
	END_IF

	gBelt.parameters.xExistBelt := TRUE;

	// This changes are done because when we have changed the reductor stops are harder than before
	// Changed from 60000 to 45000 because is not working properly in MarcoPolo (SN1).
	//29/01/2018: Dev1 with new reduction factor (15) is needed with 30000. Come back to 45000 because reductor is 35 again

	////////////////////////////////////////////////////////////
	/////BLOCK	BLOCK	BLOCK	BLOCK	BLOCK	BLOCK///////////
	////////////////////////////////////////////////////////////
	FOR iIndexBlock:=1 TO gMachine.Pt.CT.iNumBlocks DO

		gBlock[iIndexBlock].parameters.Motor.rDriveManSpeed		:=10.0;
		gBlock[iIndexBlock].parameters.Motor.rSafeMarginForwardTray:= 5.0;
		gBlock[iIndexBlock].parameters.Motor.rMinThicknessMedia:= gMachine.Pt.CT.rMinTicknessMedia;
		gBlock[iIndexBlock].parameters.Motor.rReduceSpeedDistance :=6.0;
		gBlock[iIndexBlock].parameters.Motor.rMinCleanOffsetTech := -5.0;
		gBlock[iIndexBlock].parameters.Motor.rMaxCleanOffsetTech := 0.0;
		//gBlock[iIndexBlock].parameters.Motor.rDeceleration		:= 172.5;

		gBlock[iIndexBlock].parameters.Icla.iMaxSpeedCleanMotorBwd	:=5000;
		gBlock[iIndexBlock].parameters.Icla.iMaxSpeedCleanMotorFwd	:=5000;
		gBlock[iIndexBlock].parameters.Icla.iMinSpeedCleanMotorBwd	:=300;
		gBlock[iIndexBlock].parameters.Icla.iMinSpeedCleanMotorFwd	:=300;

		gBlock[iIndexBlock].parameters.Icla.rPositionCleanMotorBwd	:= -0.5;

		gBlock[iIndexBlock].parameters.Hw.xThereIsInTraySensor	:= FALSE;
		gBlock[iIndexBlock].parameters.Hw.xIsWater	:= gMachine.St.HwData.xIsWater;

		//Time Parameters
		gBlock[iIndexBlock].parameters.tiTimeWaitTrayIn			:= T#2S;
		gBlock[iIndexBlock].parameters.tiTimeWaitTrayInAlarm 	:= T#2500ms;
		IF NOT gBlock[iIndexBlock].parameters.Hw.xIsWater THEN
			gBlock[iIndexBlock].parameters.tiTimeWaitTrayOut	:= T#5S;
			gBlock[iIndexBlock].parameters.tiTimeWaitTrayOutAlarm := T#2500ms;
		ELSE
			gBlock[iIndexBlock].parameters.tiTimeWaitTrayOut	:= T#7S;
			gBlock[iIndexBlock].parameters.tiTimeWaitTrayOutAlarm := T#7500ms;
		END_IF
		gBlock[iIndexBlock].parameters.iLastBlock:=gMachine.Pt.CT.iNumBlocks;
		gBlock[iIndexBlock].parameters.iFirstBlock:=GC_FIRST_BLOCK;

	END_FOR

	/////////////////////////////////////////////////////
	/////MODEL	MODEL	MODEL	MODEL	MODEL	MODEL////
	/////////////////////////////////////////////////////

	//By default, enable the first Block. Never a machine without a block
	gBlock[1].parameters.Hw.xExistBlock :=TRUE;

	gThicknessCtrl.parameters.sections[1].xEnabled := TRUE;
	gThicknessCtrl.parameters.iSections := gMachine.Pt.CT.iNumBlocks;

	gThicknessCtrl.parameters.Detection.ProductDetect.pMediaInProductDetectL1 := gMachine.In.ProductDetect.pPDSignalSensorL1;
	gThicknessCtrl.parameters.Detection.ProductDetect.pMediaInProductDetectL2 := gMachine.In.ProductDetect.pPDSignalSensorL2;

	// Loop all the posible blocks and assign to the block if it exists or not
	FOR iIndexBlock:=2 TO MAX_LAST_BLOCK DO

		xExistsLoopBlock := iIndexBlock <= gMachine.Pt.CT.iNumBlocks;

		//Enabling the different blocks
		gThicknessCtrl.parameters.sections[iIndexBlock].xEnabled:=xExistsLoopBlock;

		gBlock[iIndexBlock].parameters.Hw.xExistBlock:=xExistsLoopBlock;

	END_FOR

	gThicknessCtrl.parameters.rMountedMediaHeigh := 100.0;

	//Define as installed the vacuum depending on the quantity of transport vacuum of the machine
	FOR iIndexTrVacc := 1 TO MAX_LAST_TRANS_VACUUM DO
		gTransVacuum[iIndexTrVacc].Parameters.xInstalled := iIndexTrVacc <= gMachine.Pt.CT.iNumTransVacuum;
	END_FOR

	// JAM DETECTION DEVICES
	gMachine.Pt.CT.iNumSensorsPerJamDevice := 4;

END_ACTION
```
